LIN {X 0,Y 258.597,Z 623.646,A -85,B 0,C 180,E1 12291.002,E2 12291.002} C_VEL
LIN {X 0,Y 258.595,Z 623.557,A -85,B 0,C 180,E1 12285.987,E2 12285.987} C_VEL
LIN {X 0,Y 258.598,Z 623.543,A -85,B 0,C 180,E1 12281.064,E2 12281.064} C_VEL
LIN {X 0,Y 258.584,Z 623.565,A -85,B 0,C 180,E1 12276.085,E2 12276.085} C_VEL
LIN {X 0,Y 258.602,Z 623.568,A -85,B 0,C 180,E1 12271.205,E2 12271.205} C_VEL
LIN {X 0,Y 258.582,Z 623.556,A -85,B 0,C 180,E1 12268.101,E2 12268.101} C_VEL
LIN {X 0,Y 257.589,Z 623.666,A -85,B 0,C 180,E1 12266.394,E2 12266.394} C_VEL
LIN {X 0,Y 253.564,Z 624.201,A -85,B 0,C 180,E1 12263.518,E2 12263.518} C_VEL
LIN {X 0,Y 250.876,Z 624.542,A -85,B 0,C 180,E1 12261.032,E2 12261.032} C_VEL
LIN {X 0,Y 250.652,Z 624.55,A -85,B 0,C 180,E1 12260.264,E2 12260.264} C_VEL
LIN {X 0,Y 250.638,Z 624.544,A -85,B 0,C 180,E1 12255.113,E2 12255.113} C_VEL
LIN {X 0,Y 250.648,Z 624.524,A -85,B 0,C 180,E1 12250.342,E2 12250.342} C_VEL
LIN {X 0,Y 250.644,Z 624.566,A -85,B 0,C 180,E1 12245.494,E2 12245.494} C_VEL
LIN {X 0,Y 250.628,Z 624.52,A -85,B 0,C 180,E1 12240.458,E2 12240.458} C_VEL
LIN {X 0,Y 250.65,Z 624.566,A -85,B 0,C 180,E1 12235.654,E2 12235.654} C_VEL
LIN {X 0,Y 250.632,Z 624.544,A -85,B 0,C 180,E1 12230.818,E2 12230.818} C_VEL
LIN {X 0,Y 250.633,Z 624.535,A -85,B 0,C 180,E1 12225.68,E2 12225.68} C_VEL
LIN {X 0,Y 250.649,Z 624.552,A -85,B 0,C 180,E1 12220.907,E2 12220.907} C_VEL
LIN {X 0,Y 250.696,Z 624.842,A -85,B 0,C 180,E1 12216.993,E2 12216.993} C_VEL
LIN {X 0,Y 252.089,Z 628.267,A -85,B 0,C 180,E1 12215.389,E2 12215.389} C_VEL
LIN {X 0,Y 254.847,Z 634.454,A -85,B 0,C 180,E1 12212.676,E2 12212.676} C_VEL
LIN {X 0,Y 258.104,Z 641.784,A -85,B 0,C 180,E1 12209.755,E2 12209.755} C_VEL
LIN {X 0,Y 262.755,Z 653.333,A -85,B 0,C 180,E1 12205.724,E2 12205.724} C_VEL
LIN {X 0,Y 267.612,Z 666.638,A -85,B 0,C 180,E1 12201.686,E2 12201.686} C_VEL
LIN {X 0,Y 272.477,Z 681.722,A -85,B 0,C 180,E1 12197.674,E2 12197.674} C_VEL
LIN {X 0,Y 276.843,Z 696.584,A -85,B 0,C 180,E1 12194.192,E2 12194.192} C_VEL
LIN {X 0,Y 277.945,Z 699.592,A -85,B 0,C 180,E1 12193.916,E2 12193.916} C_VEL
LIN {X 0,Y 280.409,Z 735.71,A -85,B 0,C 180,E1 12192.492,E2 12192.492} C_VEL
LIN {X 0,Y 274.524,Z 880.829,A -85,B 0,C 180,E1 12188.924,E2 12188.924} C_VEL
LIN {X 0,Y 272.889,Z 899.096,A -85,B 0,C 180,E1 12188.126,E2 12188.126} C_VEL
LIN {X 0,Y 270.464,Z 916.83,A -85,B 0,C 180,E1 12186.989,E2 12186.989} C_VEL
LIN {X 0,Y 267.613,Z 933.578,A -85,B 0,C 180,E1 12185.52,E2 12185.52} C_VEL
LIN {X 0,Y 264.399,Z 949.953,A -85,B 0,C 180,E1 12183.643,E2 12183.643} C_VEL
LIN {X 0,Y 261.059,Z 965.272,A -85,B 0,C 180,E1 12181.392,E2 12181.392} C_VEL
LIN {X 0,Y 257.748,Z 979.594,A -85,B 0,C 180,E1 12178.753,E2 12178.753} C_VEL
LIN {X 0,Y 254.838,Z 992.418,A -85,B 0,C 180,E1 12175.818,E2 12175.818} C_VEL
LIN {X 0,Y 252.413,Z 1003.822,A -85,B 0,C 180,E1 12172.597,E2 12172.597} C_VEL
LIN {X 0,Y 250.561,Z 1014.181,A -85,B 0,C 180,E1 12168.961,E2 12168.961} C_VEL
LIN {X 0,Y 249.527,Z 1022.832,A -85,B 0,C 180,E1 12165.098,E2 12165.098} C_VEL
LIN {X 0,Y 249.297,Z 1029.658,A -85,B 0,C 180,E1 12161.1,E2 12161.1} C_VEL
LIN {X 0,Y 249.718,Z 1034.566,A -85,B 0,C 180,E1 12157.131,E2 12157.131} C_VEL
LIN {X 0,Y 250.306,Z 1037.499,A -85,B 0,C 180,E1 12153.436,E2 12153.436} C_VEL
LIN {X 0,Y 250.553,Z 1038.736,A -85,B 0,C 180,E1 12150.229,E2 12150.229} C_VEL
LIN {X 0,Y 250.237,Z 1038.662,A -85,B 0,C 180,E1 12147.023,E2 12147.023} C_VEL
LIN {X 0,Y 249.542,Z 1037.152,A -85,B 0,C 180,E1 12143.328,E2 12143.328} C_VEL
LIN {X 0,Y 249.014,Z 1033.682,A -85,B 0,C 180,E1 12139.122,E2 12139.122} C_VEL
LIN {X 0,Y 249.277,Z 1028.364,A -85,B 0,C 180,E1 12134.888,E2 12134.888} C_VEL
LIN {X 0,Y 250.59,Z 1021.098,A -85,B 0,C 180,E1 12130.66,E2 12130.66} C_VEL
LIN {X 0,Y 252.967,Z 1012.227,A -85,B 0,C 180,E1 12126.719,E2 12126.719} C_VEL
LIN {X 0,Y 256.245,Z 1001.804,A -85,B 0,C 180,E1 12123.088,E2 12123.088} C_VEL
LIN {X 0,Y 260.249,Z 989.873,A -85,B 0,C 180,E1 12119.782,E2 12119.782} C_VEL
LIN {X 0,Y 264.844,Z 976.404,A -85,B 0,C 180,E1 12116.81,E2 12116.81} C_VEL
LIN {X 0,Y 269.617,Z 961.83,A -85,B 0,C 180,E1 12114.262,E2 12114.262} C_VEL
LIN {X 0,Y 274.079,Z 946.842,A -85,B 0,C 180,E1 12112.203,E2 12112.203} C_VEL
LIN {X 0,Y 278.266,Z 930.98,A -85,B 0,C 180,E1 12110.507,E2 12110.507} C_VEL
LIN {X 0,Y 281.956,Z 914.615,A -85,B 0,C 180,E1 12109.177,E2 12109.177} C_VEL
LIN {X 0,Y 285.181,Z 896.361,A -85,B 0,C 180,E1 12108.103,E2 12108.103} C_VEL
LIN {X 0,Y 287.282,Z 878.288,A -85,B 0,C 180,E1 12107.378,E2 12107.378} C_VEL
LIN {X 0,Y 294.855,Z 735.141,A -85,B 0,C 180,E1 12103.879,E2 12103.879} C_VEL
LIN {X 0,Y 293.346,Z 713.913,A -85,B 0,C 180,E1 12102.776,E2 12102.776} C_VEL
LIN {X 0,Y 285.827,Z 700.894,A -85,B 0,C 180,E1 12100.524,E2 12100.524} C_VEL
LIN {X 0,Y 284.004,Z 697.557,A -85,B 0,C 180,E1 12099.847,E2 12099.847} C_VEL
LIN {X 0,Y 280.732,Z 687.562,A -85,B 0,C 180,E1 12096.244,E2 12096.244} C_VEL
LIN {X 0,Y 277.511,Z 678.838,A -85,B 0,C 180,E1 12092.468,E2 12092.468} C_VEL
LIN {X 0,Y 274.441,Z 671.373,A -85,B 0,C 180,E1 12088.507,E2 12088.507} C_VEL
LIN {X 0,Y 272.653,Z 667.299,A -85,B 0,C 180,E1 12085.873,E2 12085.873} C_VEL
LIN {X 0,Y 270.968,Z 663.499,A -85,B 0,C 180,E1 12083.025,E2 12083.025} C_VEL
LIN {X 0,Y 269.193,Z 659.526,A -85,B 0,C 180,E1 12079.303,E2 12079.303} C_VEL
LIN {X 0,Y 267.286,Z 655.366,A -85,B 0,C 180,E1 12073.19,E2 12073.19} C_VEL
LIN {X 0,Y 266.339,Z 654.288,A -85,B 0,C 180,E1 12067.984,E2 12067.984} C_VEL
LIN {X 0,Y 266.635,Z 654.723,A -85,B 0,C 180,E1 12062.579,E2 12062.579} C_VEL
LIN {X 0,Y 266.962,Z 655.866,A -85,B 0,C 180,E1 12059.962,E2 12059.962} C_VEL
LIN {X 0,Y 268.425,Z 659.327,A -85,B 0,C 180,E1 12054.656,E2 12054.656} C_VEL
LIN {X 0,Y 269.903,Z 663.428,A -85,B 0,C 180,E1 12050.619,E2 12050.619} C_VEL
LIN {X 0,Y 271.407,Z 667.48,A -85,B 0,C 180,E1 12047.446,E2 12047.446} C_VEL
LIN {X 0,Y 273.368,Z 672.921,A -85,B 0,C 180,E1 12043.86,E2 12043.86} C_VEL
LIN {X 0,Y 275.849,Z 680.778,A -85,B 0,C 180,E1 12039.636,E2 12039.636} C_VEL
LIN {X 0,Y 278.125,Z 689.309,A -85,B 0,C 180,E1 12035.805,E2 12035.805} C_VEL
LIN {X 0,Y 280.305,Z 698.744,A -85,B 0,C 180,E1 12032.141,E2 12032.141} C_VEL
LIN {X 0,Y 281.378,Z 704.237,A -85,B 0,C 180,E1 12030.283,E2 12030.283} C_VEL
LIN {X 0,Y 283.3,Z 708.755,A -85,B 0,C 180,E1 12029.527,E2 12029.527} C_VEL
LIN {X 0,Y 288.128,Z 736.946,A -85,B 0,C 180,E1 12027.253,E2 12027.253} C_VEL
LIN {X 0,Y 291.127,Z 758.877,A -85,B 0,C 180,E1 12025.756,E2 12025.756} C_VEL
LIN {X 0,Y 286.062,Z 844.009,A -85,B 0,C 180,E1 12023.499,E2 12023.499} C_VEL
LIN {X 0,Y 284.468,Z 860.29,A -85,B 0,C 180,E1 12022.719,E2 12022.719} C_VEL
LIN {X 0,Y 282.179,Z 875.724,A -85,B 0,C 180,E1 12021.636,E2 12021.636} C_VEL
LIN {X 0,Y 279.377,Z 889.681,A -85,B 0,C 180,E1 12020.305,E2 12020.305} C_VEL
LIN {X 0,Y 275.715,Z 904.283,A -85,B 0,C 180,E1 12018.476,E2 12018.476} C_VEL
LIN {X 0,Y 271.915,Z 916.881,A -85,B 0,C 180,E1 12016.418,E2 12016.418} C_VEL
LIN {X 0,Y 267.871,Z 928.54,A -85,B 0,C 180,E1 12013.969,E2 12013.969} C_VEL
LIN {X 0,Y 264.264,Z 937.852,A -85,B 0,C 180,E1 12011.462,E2 12011.462} C_VEL
LIN {X 0,Y 260.539,Z 946.484,A -85,B 0,C 180,E1 12008.44,E2 12008.44} C_VEL
LIN {X 0,Y 257.45,Z 953.125,A -85,B 0,C 180,E1 12005.355,E2 12005.355} C_VEL
LIN {X 0,Y 254.832,Z 958.272,A -85,B 0,C 180,E1 12001.984,E2 12001.984} C_VEL
LIN {X 0,Y 252.819,Z 961.87,A -85,B 0,C 180,E1 11998.332,E2 11998.332} C_VEL
LIN {X 0,Y 251.55,Z 963.593,A -85,B 0,C 180,E1 11994.667,E2 11994.667} C_VEL
LIN {X 0,Y 250.899,Z 963.561,A -85,B 0,C 180,E1 11990.773,E2 11990.773} C_VEL
LIN {X 0,Y 250.843,Z 961.794,A -85,B 0,C 180,E1 11987.155,E2 11987.155} C_VEL
LIN {X 0,Y 251.363,Z 958.066,A -85,B 0,C 180,E1 11983.339,E2 11983.339} C_VEL
LIN {X 0,Y 252.439,Z 952.682,A -85,B 0,C 180,E1 11979.806,E2 11979.806} C_VEL
LIN {X 0,Y 254.153,Z 945.316,A -85,B 0,C 180,E1 11976.324,E2 11976.324} C_VEL
LIN {X 0,Y 256.173,Z 936.954,A -85,B 0,C 180,E1 11973.356,E2 11973.356} C_VEL
LIN {X 0,Y 258.7,Z 926.457,A -85,B 0,C 180,E1 11970.442,E2 11970.442} C_VEL
LIN {X 0,Y 261.296,Z 914.754,A -85,B 0,C 180,E1 11967.916,E2 11967.916} C_VEL
LIN {X 0,Y 263.863,Z 902.135,A -85,B 0,C 180,E1 11965.762,E2 11965.762} C_VEL
LIN {X 0,Y 266.263,Z 888.571,A -85,B 0,C 180,E1 11963.964,E2 11963.964} C_VEL
LIN {X 0,Y 268.488,Z 873.21,A -85,B 0,C 180,E1 11962.403,E2 11962.403} C_VEL
LIN {X 0,Y 270.208,Z 856.922,A -85,B 0,C 180,E1 11961.22,E2 11961.22} C_VEL
LIN {X 0,Y 271.313,Z 840.68,A -85,B 0,C 180,E1 11960.434,E2 11960.434} C_VEL
LIN {X 0,Y 274.974,Z 752.221,A -85,B 0,C 180,E1 11958.038,E2 11958.038} C_VEL
LIN {X 0,Y 268.26,Z 704.82,A -85,B 0,C 180,E1 11955.593,E2 11955.593} C_VEL
LIN {X 0,Y 271.256,Z 690.293,A -85,B 0,C 180,E1 11952.628,E2 11952.628} C_VEL
LIN {X 0,Y 268.027,Z 675.976,A -85,B 0,C 180,E1 11948.556,E2 11948.556} C_VEL
LIN {X 0,Y 264.388,Z 662.466,A -85,B 0,C 180,E1 11944.328,E2 11944.328} C_VEL
LIN {X 0,Y 260.817,Z 651.102,A -85,B 0,C 180,E1 11940.361,E2 11940.361} C_VEL
LIN {X 0,Y 257.384,Z 641.549,A -85,B 0,C 180,E1 11936.639,E2 11936.639} C_VEL
LIN {X 0,Y 253.897,Z 632.375,A -85,B 0,C 180,E1 11932.665,E2 11932.665} C_VEL
LIN {X 0,Y 251.497,Z 627.253,A -85,B 0,C 180,E1 11930.113,E2 11930.113} C_VEL
LIN {X 0,Y 250.667,Z 624.683,A -85,B 0,C 180,E1 11928.733,E2 11928.733} C_VEL
LIN {X 0,Y 250.66,Z 624.573,A -85,B 0,C 180,E1 11923.78,E2 11923.78} C_VEL
LIN {X 0,Y 250.658,Z 624.548,A -85,B 0,C 180,E1 11918.935,E2 11918.935} C_VEL
LIN {X 0,Y 250.642,Z 624.527,A -85,B 0,C 180,E1 11913.925,E2 11913.925} C_VEL
LIN {X 0,Y 250.67,Z 624.564,A -85,B 0,C 180,E1 11909.12,E2 11909.12} C_VEL
LIN {X 0,Y 250.644,Z 624.533,A -85,B 0,C 180,E1 11904.261,E2 11904.261} C_VEL
LIN {X 0,Y 250.652,Z 624.55,A -85,B 0,C 180,E1 11900.264,E2 11900.264} C_VEL
LIN {X 0,Y 249.627,Z 624.66,A -85,B 0,C 180,E1 11898.503,E2 11898.503} C_VEL
LIN {X 0,Y 245.576,Z 625.199,A -85,B 0,C 180,E1 11895.536,E2 11895.536} C_VEL
LIN {X 0,Y 242.916,Z 625.539,A -85,B 0,C 180,E1 11892.968,E2 11892.968} C_VEL
LIN {X 0,Y 242.714,Z 625.55,A -85,B 0,C 180,E1 11892.174,E2 11892.174} C_VEL
LIN {X 0,Y 242.693,Z 625.518,A -85,B 0,C 180,E1 11887.1,E2 11887.1} C_VEL
LIN {X 0,Y 242.706,Z 625.517,A -85,B 0,C 180,E1 11882.125,E2 11882.125} C_VEL
LIN {X 0,Y 242.7,Z 625.559,A -85,B 0,C 180,E1 11877.167,E2 11877.167} C_VEL
LIN {X 0,Y 242.694,Z 625.517,A -85,B 0,C 180,E1 11871.948,E2 11871.948} C_VEL
LIN {X 0,Y 242.71,Z 625.533,A -85,B 0,C 180,E1 11867.147,E2 11867.147} C_VEL
LIN {X 0,Y 242.691,Z 625.567,A -85,B 0,C 180,E1 11862.121,E2 11862.121} C_VEL
LIN {X 0,Y 242.738,Z 625.842,A -85,B 0,C 180,E1 11859.569,E2 11859.569} C_VEL
LIN {X 0,Y 244.334,Z 629.512,A -85,B 0,C 180,E1 11857.631,E2 11857.631} C_VEL
LIN {X 0,Y 246.974,Z 635.346,A -85,B 0,C 180,E1 11854.844,E2 11854.844} C_VEL
LIN {X 0,Y 250.086,Z 642.133,A -85,B 0,C 180,E1 11851.851,E2 11851.851} C_VEL
LIN {X 0,Y 254.761,Z 653.796,A -85,B 0,C 180,E1 11847.474,E2 11847.474} C_VEL
LIN {X 0,Y 259.213,Z 665.715,A -85,B 0,C 180,E1 11843.557,E2 11843.557} C_VEL
LIN {X 0,Y 263.95,Z 679.981,A -85,B 0,C 180,E1 11839.485,E2 11839.485} C_VEL
LIN {X 0,Y 268.677,Z 695.94,A -85,B 0,C 180,E1 11835.454,E2 11835.454} C_VEL
LIN {X 0,Y 269.769,Z 698.685,A -85,B 0,C 180,E1 11835.085,E2 11835.085} C_VEL
LIN {X 0,Y 271.395,Z 702.547,A -85,B 0,C 180,E1 11834.732,E2 11834.732} C_VEL
LIN {X 0,Y 273.61,Z 736.548,A -85,B 0,C 180,E1 11833.358,E2 11833.358} C_VEL
LIN {X 0,Y 267.543,Z 880.121,A -85,B 0,C 180,E1 11829.757,E2 11829.757} C_VEL
LIN {X 0,Y 265.861,Z 898.397,A -85,B 0,C 180,E1 11828.943,E2 11828.943} C_VEL
LIN {X 0,Y 263.304,Z 916.451,A -85,B 0,C 180,E1 11827.759,E2 11827.759} C_VEL
LIN {X 0,Y 260.322,Z 933.306,A -85,B 0,C 180,E1 11826.238,E2 11826.238} C_VEL
LIN {X 0,Y 257.033,Z 949.39,A -85,B 0,C 180,E1 11824.337,E2 11824.337} C_VEL
LIN {X 0,Y 253.576,Z 964.616,A -85,B 0,C 180,E1 11822.033,E2 11822.033} C_VEL
LIN {X 0,Y 250.132,Z 978.897,A -85,B 0,C 180,E1 11819.32,E2 11819.32} C_VEL
LIN {X 0,Y 247.002,Z 992.117,A -85,B 0,C 180,E1 11816.183,E2 11816.183} C_VEL
LIN {X 0,Y 244.504,Z 1003.394,A -85,B 0,C 180,E1 11812.861,E2 11812.861} C_VEL
LIN {X 0,Y 242.657,Z 1013.28,A -85,B 0,C 180,E1 11809.247,E2 11809.247} C_VEL
LIN {X 0,Y 241.594,Z 1021.695,A -85,B 0,C 180,E1 11805.358,E2 11805.358} C_VEL
LIN {X 0,Y 241.341,Z 1028.525,A -85,B 0,C 180,E1 11801.229,E2 11801.229} C_VEL
LIN {X 0,Y 241.743,Z 1033.199,A -85,B 0,C 180,E1 11797.367,E2 11797.367} C_VEL
LIN {X 0,Y 242.371,Z 1036.215,A -85,B 0,C 180,E1 11793.548,E2 11793.548} C_VEL
LIN {X 0,Y 242.65,Z 1037.49,A -85,B 0,C 180,E1 11790.237,E2 11790.237} C_VEL
LIN {X 0,Y 242.298,Z 1037.466,A -85,B 0,C 180,E1 11786.925,E2 11786.925} C_VEL
LIN {X 0,Y 241.553,Z 1035.998,A -85,B 0,C 180,E1 11783.106,E2 11783.106} C_VEL
LIN {X 0,Y 241.028,Z 1032.576,A -85,B 0,C 180,E1 11778.757,E2 11778.757} C_VEL
LIN {X 0,Y 241.377,Z 1027.303,A -85,B 0,C 180,E1 11774.381,E2 11774.381} C_VEL
LIN {X 0,Y 242.847,Z 1020.08,A -85,B 0,C 180,E1 11770.018,E2 11770.018} C_VEL
LIN {X 0,Y 245.429,Z 1011.278,A -85,B 0,C 180,E1 11765.959,E2 11765.959} C_VEL
LIN {X 0,Y 248.944,Z 1000.915,A -85,B 0,C 180,E1 11762.232,E2 11762.232} C_VEL
LIN {X 0,Y 253.202,Z 989.077,A -85,B 0,C 180,E1 11758.849,E2 11758.849} C_VEL
LIN {X 0,Y 258.054,Z 975.679,A -85,B 0,C 180,E1 11755.819,E2 11755.819} C_VEL
LIN {X 0,Y 262.846,Z 961.787,A -85,B 0,C 180,E1 11753.329,E2 11753.329} C_VEL
LIN {X 0,Y 267.494,Z 947.056,A -85,B 0,C 180,E1 11751.238,E2 11751.238} C_VEL
LIN {X 0,Y 271.841,Z 931.515,A -85,B 0,C 180,E1 11749.52,E2 11749.52} C_VEL
LIN {X 0,Y 275.737,Z 915.143,A -85,B 0,C 180,E1 11748.148,E2 11748.148} C_VEL
LIN {X 0,Y 279.04,Z 897.565,A -85,B 0,C 180,E1 11747.076,E2 11747.076} C_VEL
LIN {X 0,Y 281.38,Z 879.001,A -85,B 0,C 180,E1 11746.298,E2 11746.298} C_VEL
LIN {X 0,Y 283.499,Z 842.829,A -85,B 0,C 180,E1 11745.373,E2 11745.373} C_VEL
LIN {X 0,Y 289.419,Z 736.279,A -85,B 0,C 180,E1 11742.745,E2 11742.745} C_VEL
LIN {X 0,Y 288.201,Z 717.926,A -85,B 0,C 180,E1 11741.767,E2 11741.767} C_VEL
LIN {X 0,Y 280.288,Z 704.05,A -85,B 0,C 180,E1 11739.252,E2 11739.252} C_VEL
LIN {X 0,Y 276.518,Z 697.804,A -85,B 0,C 180,E1 11737.831,E2 11737.831} C_VEL
LIN {X 0,Y 273.304,Z 688.322,A -85,B 0,C 180,E1 11734.037,E2 11734.037} C_VEL
LIN {X 0,Y 270.315,Z 680.495,A -85,B 0,C 180,E1 11730.201,E2 11730.201} C_VEL
LIN {X 0,Y 267.774,Z 674.014,A -85,B 0,C 180,E1 11726.343,E2 11726.343} C_VEL
LIN {X 0,Y 265.6,Z 669.326,A -85,B 0,C 180,E1 11722.734,E2 11722.734} C_VEL
LIN {X 0,Y 263.921,Z 665.479,A -85,B 0,C 180,E1 11719.014,E2 11719.014} C_VEL
LIN {X 0,Y 262.121,Z 661.451,A -85,B 0,C 180,E1 11713.006,E2 11713.006} C_VEL
LIN {X 0,Y 261.19,Z 660.419,A -85,B 0,C 180,E1 11707.699,E2 11707.699} C_VEL
LIN {X 0,Y 261.503,Z 660.871,A -85,B 0,C 180,E1 11702.41,E2 11702.41} C_VEL
LIN {X 0,Y 261.784,Z 662.197,A -85,B 0,C 180,E1 11699.562,E2 11699.562} C_VEL
LIN {X 0,Y 263.055,Z 665.27,A -85,B 0,C 180,E1 11694.766,E2 11694.766} C_VEL
LIN {X 0,Y 264.418,Z 669.141,A -85,B 0,C 180,E1 11690.861,E2 11690.861} C_VEL
LIN {X 0,Y 265.807,Z 673.148,A -85,B 0,C 180,E1 11687.619,E2 11687.619} C_VEL
LIN {X 0,Y 267.58,Z 678.248,A -85,B 0,C 180,E1 11684.17,E2 11684.17} C_VEL
LIN {X 0,Y 269.926,Z 686.085,A -85,B 0,C 180,E1 11679.849,E2 11679.849} C_VEL
LIN {X 0,Y 272.082,Z 694.639,A -85,B 0,C 180,E1 11675.926,E2 11675.926} C_VEL
LIN {X 0,Y 274.146,Z 703.986,A -85,B 0,C 180,E1 11672.288,E2 11672.288} C_VEL
LIN {X 0,Y 278.578,Z 712.773,A -85,B 0,C 180,E1 11670.576,E2 11670.576} C_VEL
LIN {X 0,Y 283.059,Z 740.327,A -85,B 0,C 180,E1 11668.302,E2 11668.302} C_VEL
LIN {X 0,Y 285.641,Z 760.611,A -85,B 0,C 180,E1 11666.891,E2 11666.891} C_VEL
LIN {X 0,Y 280.42,Z 844.7,A -85,B 0,C 180,E1 11664.638,E2 11664.638} C_VEL
LIN {X 0,Y 278.743,Z 861.013,A -85,B 0,C 180,E1 11663.847,E2 11663.847} C_VEL
LIN {X 0,Y 276.339,Z 876.45,A -85,B 0,C 180,E1 11662.751,E2 11662.751} C_VEL
LIN {X 0,Y 273.247,Z 891.044,A -85,B 0,C 180,E1 11661.333,E2 11661.333} C_VEL
LIN {X 0,Y 269.472,Z 905.321,A -85,B 0,C 180,E1 11659.508,E2 11659.508} C_VEL
LIN {X 0,Y 265.498,Z 917.826,A -85,B 0,C 180,E1 11657.43,E2 11657.43} C_VEL
LIN {X 0,Y 261.197,Z 929.61,A -85,B 0,C 180,E1 11654.912,E2 11654.912} C_VEL
LIN {X 0,Y 257.246,Z 939.243,A -85,B 0,C 180,E1 11652.253,E2 11652.253} C_VEL
LIN {X 0,Y 253.322,Z 947.821,A -85,B 0,C 180,E1 11649.162,E2 11649.162} C_VEL
LIN {X 0,Y 250.053,Z 954.415,A -85,B 0,C 180,E1 11646,E2 11646} C_VEL
LIN {X 0,Y 247.261,Z 959.53,A -85,B 0,C 180,E1 11642.535,E2 11642.535} C_VEL
LIN {X 0,Y 245.063,Z 963.168,A -85,B 0,C 180,E1 11638.692,E2 11638.692} C_VEL
LIN {X 0,Y 243.71,Z 964.821,A -85,B 0,C 180,E1 11634.947,E2 11634.947} C_VEL
LIN {X 0,Y 242.997,Z 964.762,A -85,B 0,C 180,E1 11630.925,E2 11630.925} C_VEL
LIN {X 0,Y 242.917,Z 963.009,A -85,B 0,C 180,E1 11627.238,E2 11627.238} C_VEL
LIN {X 0,Y 243.451,Z 959.239,A -85,B 0,C 180,E1 11623.251,E2 11623.251} C_VEL
LIN {X 0,Y 244.551,Z 953.938,A -85,B 0,C 180,E1 11619.65,E2 11619.65} C_VEL
LIN {X 0,Y 246.336,Z 946.564,A -85,B 0,C 180,E1 11616.04,E2 11616.04} C_VEL
LIN {X 0,Y 248.423,Z 938.304,A -85,B 0,C 180,E1 11612.999,E2 11612.999} C_VEL
LIN {X 0,Y 251.042,Z 927.866,A -85,B 0,C 180,E1 11610,E2 11610} C_VEL
LIN {X 0,Y 253.744,Z 916.28,A -85,B 0,C 180,E1 11607.402,E2 11607.402} C_VEL
LIN {X 0,Y 256.545,Z 903.091,A -85,B 0,C 180,E1 11605.081,E2 11605.081} C_VEL
LIN {X 0,Y 259.046,Z 889.548,A -85,B 0,C 180,E1 11603.239,E2 11603.239} C_VEL
LIN {X 0,Y 261.363,Z 874.224,A -85,B 0,C 180,E1 11601.641,E2 11601.641} C_VEL
LIN {X 0,Y 263.149,Z 858.159,A -85,B 0,C 180,E1 11600.438,E2 11600.438} C_VEL
LIN {X 0,Y 264.344,Z 841.574,A -85,B 0,C 180,E1 11599.606,E2 11599.606} C_VEL
LIN {X 0,Y 268.14,Z 753.168,A -85,B 0,C 180,E1 11597.16,E2 11597.16} C_VEL
LIN {X 0,Y 261.435,Z 704.987,A -85,B 0,C 180,E1 11594.599,E2 11594.599} C_VEL
LIN {X 0,Y 262.769,Z 698.408,A -85,B 0,C 180,E1 11593.304,E2 11593.304} C_VEL
LIN {X 0,Y 263.977,Z 692.922,A -85,B 0,C 180,E1 11592.133,E2 11592.133} C_VEL
LIN {X 0,Y 260.89,Z 678.952,A -85,B 0,C 180,E1 11588.044,E2 11588.044} C_VEL
LIN {X 0,Y 257.331,Z 665.522,A -85,B 0,C 180,E1 11583.707,E2 11583.707} C_VEL
LIN {X 0,Y 253.626,Z 653.753,A -85,B 0,C 180,E1 11579.432,E2 11579.432} C_VEL
LIN {X 0,Y 250.169,Z 643.88,A -85,B 0,C 180,E1 11575.42,E2 11575.42} C_VEL
LIN {X 0,Y 246.898,Z 635.905,A -85,B 0,C 180,E1 11571.712,E2 11571.712} C_VEL
LIN {X 0,Y 244.349,Z 629.521,A -85,B 0,C 180,E1 11568.478,E2 11568.478} C_VEL
LIN {X 0,Y 242.732,Z 625.669,A -85,B 0,C 180,E1 11566.209,E2 11566.209} C_VEL
LIN {X 0,Y 242.72,Z 625.52,A -85,B 0,C 180,E1 11561.074,E2 11561.074} C_VEL
LIN {X 0,Y 242.706,Z 625.539,A -85,B 0,C 180,E1 11556.094,E2 11556.094} C_VEL
LIN {X 0,Y 242.73,Z 625.546,A -85,B 0,C 180,E1 11550.992,E2 11550.992} C_VEL
LIN {X 0,Y 242.699,Z 625.508,A -85,B 0,C 180,E1 11545.894,E2 11545.894} C_VEL
LIN {X 0,Y 242.722,Z 625.548,A -85,B 0,C 180,E1 11540.749,E2 11540.749} C_VEL
LIN {X 0,Y 242.699,Z 625.518,A -85,B 0,C 180,E1 11535.778,E2 11535.778} C_VEL
LIN {X 0,Y 242.714,Z 625.55,A -85,B 0,C 180,E1 11532.174,E2 11532.174} C_VEL
LIN {X 0,Y 241.849,Z 625.639,A -85,B 0,C 180,E1 11530.484,E2 11530.484} C_VEL
LIN {X 0,Y 238.401,Z 626.094,A -85,B 0,C 180,E1 11527.806,E2 11527.806} C_VEL
LIN {X 0,Y 235.052,Z 626.521,A -85,B 0,C 180,E1 11524.771,E2 11524.771} C_VEL
LIN {X 0,Y 234.769,Z 626.539,A -85,B 0,C 180,E1 11523.813,E2 11523.813} C_VEL
LIN {X 0,Y 234.748,Z 626.514,A -85,B 0,C 180,E1 11518.536,E2 11518.536} C_VEL
LIN {X 0,Y 234.776,Z 626.502,A -85,B 0,C 180,E1 11513.398,E2 11513.398} C_VEL
LIN {X 0,Y 234.751,Z 626.542,A -85,B 0,C 180,E1 11508.204,E2 11508.204} C_VEL
LIN {X 0,Y 234.776,Z 626.571,A -85,B 0,C 180,E1 11503.167,E2 11503.167} C_VEL
LIN {X 0,Y 234.844,Z 627.105,A -85,B 0,C 180,E1 11502.405,E2 11502.405} C_VEL
LIN {X 0,Y 237.219,Z 632.279,A -85,B 0,C 180,E1 11499.346,E2 11499.346} C_VEL
LIN {X 0,Y 239.171,Z 636.504,A -85,B 0,C 180,E1 11497.121,E2 11497.121} C_VEL
LIN {X 0,Y 241.374,Z 641.447,A -85,B 0,C 180,E1 11494.744,E2 11494.744} C_VEL
LIN {X 0,Y 244.203,Z 647.836,A -85,B 0,C 180,E1 11491.911,E2 11491.911} C_VEL
LIN {X 0,Y 248.35,Z 658.225,A -85,B 0,C 180,E1 11487.898,E2 11487.898} C_VEL
LIN {X 0,Y 252.84,Z 670.501,A -85,B 0,C 180,E1 11483.778,E2 11483.778} C_VEL
LIN {X 0,Y 257.354,Z 684.492,A -85,B 0,C 180,E1 11479.694,E2 11479.694} C_VEL
LIN {X 0,Y 261.13,Z 697.26,A -85,B 0,C 180,E1 11476.432,E2 11476.432} C_VEL
LIN {X 0,Y 264.867,Z 705.427,A -85,B 0,C 180,E1 11475.581,E2 11475.581} C_VEL
LIN {X 0,Y 266.844,Z 737.351,A -85,B 0,C 180,E1 11474.256,E2 11474.256} C_VEL
LIN {X 0,Y 260.576,Z 879.607,A -85,B 0,C 180,E1 11470.617,E2 11470.617} C_VEL
LIN {X 0,Y 258.847,Z 897.838,A -85,B 0,C 180,E1 11469.786,E2 11469.786} C_VEL
LIN {X 0,Y 256.191,Z 915.969,A -85,B 0,C 180,E1 11468.571,E2 11468.571} C_VEL
LIN {X 0,Y 253.172,Z 932.478,A -85,B 0,C 180,E1 11467.048,E2 11467.048} C_VEL
LIN {X 0,Y 249.705,Z 948.809,A -85,B 0,C 180,E1 11465.072,E2 11465.072} C_VEL
LIN {X 0,Y 246.117,Z 963.992,A -85,B 0,C 180,E1 11462.706,E2 11462.706} C_VEL
LIN {X 0,Y 242.542,Z 978.199,A -85,B 0,C 180,E1 11459.922,E2 11459.922} C_VEL
LIN {X 0,Y 239.39,Z 990.916,A -85,B 0,C 180,E1 11456.814,E2 11456.814} C_VEL
LIN {X 0,Y 236.758,Z 1002.217,A -85,B 0,C 180,E1 11453.39,E2 11453.39} C_VEL
LIN {X 0,Y 234.802,Z 1012.118,A -85,B 0,C 180,E1 11449.659,E2 11449.659} C_VEL
LIN {X 0,Y 233.663,Z 1020.54,A -85,B 0,C 180,E1 11445.64,E2 11445.64} C_VEL
LIN {X 0,Y 233.386,Z 1027.373,A -85,B 0,C 180,E1 11441.366,E2 11441.366} C_VEL
LIN {X 0,Y 233.846,Z 1032.268,A -85,B 0,C 180,E1 11437.123,E2 11437.123} C_VEL
LIN {X 0,Y 234.513,Z 1035.165,A -85,B 0,C 180,E1 11433.178,E2 11433.178} C_VEL
LIN {X 0,Y 234.729,Z 1036.351,A -85,B 0,C 180,E1 11429.756,E2 11429.756} C_VEL
LIN {X 0,Y 234.261,Z 1036.177,A -85,B 0,C 180,E1 11426.33,E2 11426.33} C_VEL
LIN {X 0,Y 233.431,Z 1034.406,A -85,B 0,C 180,E1 11422.122,E2 11422.122} C_VEL
LIN {X 0,Y 233.047,Z 1030.736,A -85,B 0,C 180,E1 11417.613,E2 11417.613} C_VEL
LIN {X 0,Y 233.67,Z 1025.211,A -85,B 0,C 180,E1 11413.084,E2 11413.084} C_VEL
LIN {X 0,Y 235.399,Z 1018.167,A -85,B 0,C 180,E1 11408.836,E2 11408.836} C_VEL
LIN {X 0,Y 238.347,Z 1009.151,A -85,B 0,C 180,E1 11404.667,E2 11404.667} C_VEL
LIN {X 0,Y 242.251,Z 998.612,A -85,B 0,C 180,E1 11400.855,E2 11400.855} C_VEL
LIN {X 0,Y 246.904,Z 986.545,A -85,B 0,C 180,E1 11397.412,E2 11397.412} C_VEL
LIN {X 0,Y 251.992,Z 973.282,A -85,B 0,C 180,E1 11394.429,E2 11394.429} C_VEL
LIN {X 0,Y 257.037,Z 959.234,A -85,B 0,C 180,E1 11391.935,E2 11391.935} C_VEL
LIN {X 0,Y 261.956,Z 944.077,A -85,B 0,C 180,E1 11389.83,E2 11389.83} C_VEL
LIN {X 0,Y 266.55,Z 928.045,A -85,B 0,C 180,E1 11388.111,E2 11388.111} C_VEL
LIN {X 0,Y 270.646,Z 911.008,A -85,B 0,C 180,E1 11386.741,E2 11386.741} C_VEL
LIN {X 0,Y 273.902,Z 893.411,A -85,B 0,C 180,E1 11385.722,E2 11385.722} C_VEL
LIN {X 0,Y 276.085,Z 875.179,A -85,B 0,C 180,E1 11385.005,E2 11385.005} C_VEL
LIN {X 0,Y 284.098,Z 737.345,A -85,B 0,C 180,E1 11381.564,E2 11381.564} C_VEL
LIN {X 0,Y 283.153,Z 721.957,A -85,B 0,C 180,E1 11380.721,E2 11380.721} C_VEL
LIN {X 0,Y 276.319,Z 709.752,A -85,B 0,C 180,E1 11378.424,E2 11378.424} C_VEL
LIN {X 0,Y 269.165,Z 698.327,A -85,B 0,C 180,E1 11375.676,E2 11375.676} C_VEL
LIN {X 0,Y 266.21,Z 689.866,A -85,B 0,C 180,E1 11371.915,E2 11371.915} C_VEL
LIN {X 0,Y 263.35,Z 682.543,A -85,B 0,C 180,E1 11367.839,E2 11367.839} C_VEL
LIN {X 0,Y 261.62,Z 678.487,A -85,B 0,C 180,E1 11365.074,E2 11365.074} C_VEL
LIN {X 0,Y 260.333,Z 675.308,A -85,B 0,C 180,E1 11362.586,E2 11362.586} C_VEL
LIN {X 0,Y 258.749,Z 671.574,A -85,B 0,C 180,E1 11358.94,E2 11358.94} C_VEL
LIN {X 0,Y 256.984,Z 667.562,A -85,B 0,C 180,E1 11352.813,E2 11352.813} C_VEL
LIN {X 0,Y 256.072,Z 666.567,A -85,B 0,C 180,E1 11347.357,E2 11347.357} C_VEL
LIN {X 0,Y 256.422,Z 667.088,A -85,B 0,C 180,E1 11342.011,E2 11342.011} C_VEL
LIN {X 0,Y 257.691,Z 671.016,A -85,B 0,C 180,E1 11335.103,E2 11335.103} C_VEL
LIN {X 0,Y 258.972,Z 675.105,A -85,B 0,C 180,E1 11330.892,E2 11330.892} C_VEL
LIN {X 0,Y 260.222,Z 678.826,A -85,B 0,C 180,E1 11327.799,E2 11327.799} C_VEL
LIN {X 0,Y 261.927,Z 684.175,A -85,B 0,C 180,E1 11324.146,E2 11324.146} C_VEL
LIN {X 0,Y 264.009,Z 691.401,A -85,B 0,C 180,E1 11320.071,E2 11320.071} C_VEL
LIN {X 0,Y 266.146,Z 700.299,A -85,B 0,C 180,E1 11315.909,E2 11315.909} C_VEL
LIN {X 0,Y 267.11,Z 704.257,A -85,B 0,C 180,E1 11314.383,E2 11314.383} C_VEL
LIN {X 0,Y 273.705,Z 716.398,A -85,B 0,C 180,E1 11311.766,E2 11311.766} C_VEL
LIN {X 0,Y 274.402,Z 719.247,A -85,B 0,C 180,E1 11311.44,E2 11311.44} C_VEL
LIN {X 0,Y 278.53,Z 746.876,A -85,B 0,C 180,E1 11309.143,E2 11309.143} C_VEL
LIN {X 0,Y 280.276,Z 762.256,A -85,B 0,C 180,E1 11308.073,E2 11308.073} C_VEL
LIN {X 0,Y 274.892,Z 845.39,A -85,B 0,C 180,E1 11305.823,E2 11305.823} C_VEL
LIN {X 0,Y 273.132,Z 861.754,A -85,B 0,C 180,E1 11305.022,E2 11305.022} C_VEL
LIN {X 0,Y 270.508,Z 877.805,A -85,B 0,C 180,E1 11303.864,E2 11303.864} C_VEL
LIN {X 0,Y 267.252,Z 892.337,A -85,B 0,C 180,E1 11302.422,E2 11302.422} C_VEL
LIN {X 0,Y 263.364,Z 906.337,A -85,B 0,C 180,E1 11300.604,E2 11300.604} C_VEL
LIN {X 0,Y 259.135,Z 918.995,A -85,B 0,C 180,E1 11298.464,E2 11298.464} C_VEL
LIN {X 0,Y 254.653,Z 930.613,A -85,B 0,C 180,E1 11295.932,E2 11295.932} C_VEL
LIN {X 0,Y 250.632,Z 939.926,A -85,B 0,C 180,E1 11293.327,E2 11293.327} C_VEL
LIN {X 0,Y 246.442,Z 948.57,A -85,B 0,C 180,E1 11290.172,E2 11290.172} C_VEL
LIN {X 0,Y 242.687,Z 955.705,A -85,B 0,C 180,E1 11286.683,E2 11286.683} C_VEL
LIN {X 0,Y 239.533,Z 961.081,A -85,B 0,C 180,E1 11282.864,E2 11282.864} C_VEL
LIN {X 0,Y 237.274,Z 964.518,A -85,B 0,C 180,E1 11278.986,E2 11278.986} C_VEL
LIN {X 0,Y 235.761,Z 966.125,A -85,B 0,C 180,E1 11274.825,E2 11274.825} C_VEL
LIN {X 0,Y 235.082,Z 965.929,A -85,B 0,C 180,E1 11270.932,E2 11270.932} C_VEL
LIN {X 0,Y 235.018,Z 963.851,A -85,B 0,C 180,E1 11266.814,E2 11266.814} C_VEL
LIN {X 0,Y 235.575,Z 960.224,A -85,B 0,C 180,E1 11263,E2 11263} C_VEL
LIN {X 0,Y 236.761,Z 954.743,A -85,B 0,C 180,E1 11259.234,E2 11259.234} C_VEL
LIN {X 0,Y 238.499,Z 947.861,A -85,B 0,C 180,E1 11255.774,E2 11255.774} C_VEL
LIN {X 0,Y 240.677,Z 939.614,A -85,B 0,C 180,E1 11252.619,E2 11252.619} C_VEL
LIN {X 0,Y 243.394,Z 929.224,A -85,B 0,C 180,E1 11249.529,E2 11249.529} C_VEL
LIN {X 0,Y 246.207,Z 917.743,A -85,B 0,C 180,E1 11246.857,E2 11246.857} C_VEL
LIN {X 0,Y 249.135,Z 904.538,A -85,B 0,C 180,E1 11244.452,E2 11244.452} C_VEL
LIN {X 0,Y 251.709,Z 891.341,A -85,B 0,C 180,E1 11242.582,E2 11242.582} C_VEL
LIN {X 0,Y 254.156,Z 875.945,A -85,B 0,C 180,E1 11240.914,E2 11240.914} C_VEL
LIN {X 0,Y 256.032,Z 860.295,A -85,B 0,C 180,E1 11239.679,E2 11239.679} C_VEL
LIN {X 0,Y 257.371,Z 843.117,A -85,B 0,C 180,E1 11238.771,E2 11238.771} C_VEL
LIN {X 0,Y 261.466,Z 756.463,A -85,B 0,C 180,E1 11236.337,E2 11236.337} C_VEL
LIN {X 0,Y 255.462,Z 710.739,A -85,B 0,C 180,E1 11233.88,E2 11233.88} C_VEL
LIN {X 0,Y 254.685,Z 704.29,A -85,B 0,C 180,E1 11233.463,E2 11233.463} C_VEL
LIN {X 0,Y 256.716,Z 695.552,A -85,B 0,C 180,E1 11231.61,E2 11231.61} C_VEL
LIN {X 0,Y 253.776,Z 682.019,A -85,B 0,C 180,E1 11227.531,E2 11227.531} C_VEL
LIN {X 0,Y 250.551,Z 669.499,A -85,B 0,C 180,E1 11223.369,E2 11223.369} C_VEL
LIN {X 0,Y 246.77,Z 657.142,A -85,B 0,C 180,E1 11218.753,E2 11218.753} C_VEL
LIN {X 0,Y 243.458,Z 647.865,A -85,B 0,C 180,E1 11214.814,E2 11214.814} C_VEL
LIN {X 0,Y 239.947,Z 638.608,A -85,B 0,C 180,E1 11210.39,E2 11210.39} C_VEL
LIN {X 0,Y 236.538,Z 630.666,A -85,B 0,C 180,E1 11205.94,E2 11205.94} C_VEL
LIN {X 0,Y 234.794,Z 626.655,A -85,B 0,C 180,E1 11203.264,E2 11203.264} C_VEL
LIN {X 0,Y 234.769,Z 626.541,A -85,B 0,C 180,E1 11198.138,E2 11198.138} C_VEL
LIN {X 0,Y 234.778,Z 626.503,A -85,B 0,C 180,E1 11192.967,E2 11192.967} C_VEL
LIN {X 0,Y 234.764,Z 626.514,A -85,B 0,C 180,E1 11187.937,E2 11187.937} C_VEL
LIN {X 0,Y 234.788,Z 626.535,A -85,B 0,C 180,E1 11182.801,E2 11182.801} C_VEL
LIN {X 0,Y 234.755,Z 626.492,A -85,B 0,C 180,E1 11177.602,E2 11177.602} C_VEL
LIN {X 0,Y 234.775,Z 626.546,A -85,B 0,C 180,E1 11172.545,E2 11172.545} C_VEL
LIN {X 0,Y 234.756,Z 626.502,A -85,B 0,C 180,E1 11167.342,E2 11167.342} C_VEL
LIN {X 0,Y 234.769,Z 626.539,A -85,B 0,C 180,E1 11163.813,E2 11163.813} C_VEL
LIN {X 0,Y 233.897,Z 626.626,A -85,B 0,C 180,E1 11162.066,E2 11162.066} C_VEL
LIN {X 0,Y 230.463,Z 627.071,A -85,B 0,C 180,E1 11159.295,E2 11159.295} C_VEL
LIN {X 0,Y 227.116,Z 627.505,A -85,B 0,C 180,E1 11156.154,E2 11156.154} C_VEL
LIN {X 0,Y 226.82,Z 627.517,A -85,B 0,C 180,E1 11155.162,E2 11155.162} C_VEL
LIN {X 0,Y 226.821,Z 627.525,A -85,B 0,C 180,E1 11149.845,E2 11149.845} C_VEL
LIN {X 0,Y 226.852,Z 627.813,A -85,B 0,C 180,E1 11146.004,E2 11146.004} C_VEL
LIN {X 0,Y 228.721,Z 631.795,A -85,B 0,C 180,E1 11143.212,E2 11143.212} C_VEL
LIN {X 0,Y 231.382,Z 637.458,A -85,B 0,C 180,E1 11139.776,E2 11139.776} C_VEL
LIN {X 0,Y 233.571,Z 642.529,A -85,B 0,C 180,E1 11137.074,E2 11137.074} C_VEL
LIN {X 0,Y 236.529,Z 649.009,A -85,B 0,C 180,E1 11133.92,E2 11133.92} C_VEL
LIN {X 0,Y 240.51,Z 658.784,A -85,B 0,C 180,E1 11129.8,E2 11129.8} C_VEL
LIN {X 0,Y 244.964,Z 670.919,A -85,B 0,C 180,E1 11125.435,E2 11125.435} C_VEL
LIN {X 0,Y 249.314,Z 684.221,A -85,B 0,C 180,E1 11121.272,E2 11121.272} C_VEL
LIN {X 0,Y 253.275,Z 697.424,A -85,B 0,C 180,E1 11117.695,E2 11117.695} C_VEL
LIN {X 0,Y 258.394,Z 708.243,A -85,B 0,C 180,E1 11116.477,E2 11116.477} C_VEL
LIN {X 0,Y 260.144,Z 738.2,A -85,B 0,C 180,E1 11115.2,E2 11115.2} C_VEL
LIN {X 0,Y 253.674,Z 878.901,A -85,B 0,C 180,E1 11111.525,E2 11111.525} C_VEL
LIN {X 0,Y 251.89,Z 897.143,A -85,B 0,C 180,E1 11110.677,E2 11110.677} C_VEL
LIN {X 0,Y 249.244,Z 914.685,A -85,B 0,C 180,E1 11109.483,E2 11109.483} C_VEL
LIN {X 0,Y 245.992,Z 931.928,A -85,B 0,C 180,E1 11107.862,E2 11107.862} C_VEL
LIN {X 0,Y 242.42,Z 948.096,A -85,B 0,C 180,E1 11105.852,E2 11105.852} C_VEL
LIN {X 0,Y 238.69,Z 963.3,A -85,B 0,C 180,E1 11103.418,E2 11103.418} C_VEL
LIN {X 0,Y 234.981,Z 977.456,A -85,B 0,C 180,E1 11100.563,E2 11100.563} C_VEL
LIN {X 0,Y 231.584,Z 990.602,A -85,B 0,C 180,E1 11097.236,E2 11097.236} C_VEL
LIN {X 0,Y 228.865,Z 1001.788,A -85,B 0,C 180,E1 11093.699,E2 11093.699} C_VEL
LIN {X 0,Y 226.853,Z 1011.553,A -85,B 0,C 180,E1 11089.84,E2 11089.84} C_VEL
LIN {X 0,Y 225.695,Z 1019.829,A -85,B 0,C 180,E1 11085.679,E2 11085.679} C_VEL
LIN {X 0,Y 225.44,Z 1026.554,A -85,B 0,C 180,E1 11081.254,E2 11081.254} C_VEL
LIN {X 0,Y 225.955,Z 1031.337,A -85,B 0,C 180,E1 11076.862,E2 11076.862} C_VEL
LIN {X 0,Y 226.618,Z 1033.992,A -85,B 0,C 180,E1 11073.035,E2 11073.035} C_VEL
LIN {X 0,Y 226.826,Z 1035.1,A -85,B 0,C 180,E1 11069.748,E2 11069.748} C_VEL
LIN {X 0,Y 226.31,Z 1034.979,A -85,B 0,C 180,E1 11066.201,E2 11066.201} C_VEL
LIN {X 0,Y 225.43,Z 1033.251,A -85,B 0,C 180,E1 11061.841,E2 11061.841} C_VEL
LIN {X 0,Y 225.088,Z 1029.626,A -85,B 0,C 180,E1 11057.168,E2 11057.168} C_VEL
LIN {X 0,Y 225.829,Z 1024.158,A -85,B 0,C 180,E1 11052.478,E2 11052.478} C_VEL
LIN {X 0,Y 227.902,Z 1016.725,A -85,B 0,C 180,E1 11047.834,E2 11047.834} C_VEL
LIN {X 0,Y 231.163,Z 1007.648,A -85,B 0,C 180,E1 11043.544,E2 11043.544} C_VEL
LIN {X 0,Y 235.412,Z 997.038,A -85,B 0,C 180,E1 11039.641,E2 11039.641} C_VEL
LIN {X 0,Y 240.413,Z 984.886,A -85,B 0,C 180,E1 11036.131,E2 11036.131} C_VEL
LIN {X 0,Y 245.787,Z 971.635,A -85,B 0,C 180,E1 11033.128,E2 11033.128} C_VEL
LIN {X 0,Y 251.309,Z 956.899,A -85,B 0,C 180,E1 11030.52,E2 11030.52} C_VEL
LIN {X 0,Y 256.349,Z 942.01,A -85,B 0,C 180,E1 11028.466,E2 11028.466} C_VEL
LIN {X 0,Y 261.168,Z 925.715,A -85,B 0,C 180,E1 11026.742,E2 11026.742} C_VEL
LIN {X 0,Y 265.213,Z 909.272,A -85,B 0,C 180,E1 11025.441,E2 11025.441} C_VEL
LIN {X 0,Y 268.572,Z 891.452,A -85,B 0,C 180,E1 11024.426,E2 11024.426} C_VEL
LIN {X 0,Y 270.713,Z 873.229,A -85,B 0,C 180,E1 11023.732,E2 11023.732} C_VEL
LIN {X 0,Y 278.9,Z 738.276,A -85,B 0,C 180,E1 11020.331,E2 11020.331} C_VEL
LIN {X 0,Y 278.212,Z 725.906,A -85,B 0,C 180,E1 11019.636,E2 11019.636} C_VEL
LIN {X 0,Y 271.604,Z 714.193,A -85,B 0,C 180,E1 11017.27,E2 11017.27} C_VEL
LIN {X 0,Y 264.718,Z 703.383,A -85,B 0,C 180,E1 11014.57,E2 11014.57} C_VEL
LIN {X 0,Y 261.59,Z 698.338,A -85,B 0,C 180,E1 11013.067,E2 11013.067} C_VEL
LIN {X 0,Y 258.664,Z 690.431,A -85,B 0,C 180,E1 11008.893,E2 11008.893} C_VEL
LIN {X 0,Y 256.436,Z 684.705,A -85,B 0,C 180,E1 11005.15,E2 11005.15} C_VEL
LIN {X 0,Y 254.953,Z 681.101,A -85,B 0,C 180,E1 11002.252,E2 11002.252} C_VEL
LIN {X 0,Y 253.458,Z 677.5,A -85,B 0,C 180,E1 10998.634,E2 10998.634} C_VEL
LIN {X 0,Y 251.878,Z 673.728,A -85,B 0,C 180,E1 10992.844,E2 10992.844} C_VEL
LIN {X 0,Y 250.949,Z 672.711,A -85,B 0,C 180,E1 10987.325,E2 10987.325} C_VEL
LIN {X 0,Y 251.243,Z 673.183,A -85,B 0,C 180,E1 10982.052,E2 10982.052} C_VEL
LIN {X 0,Y 252.351,Z 676.98,A -85,B 0,C 180,E1 10975.227,E2 10975.227} C_VEL
LIN {X 0,Y 253.484,Z 680.809,A -85,B 0,C 180,E1 10971.15,E2 10971.15} C_VEL
LIN {X 0,Y 254.655,Z 684.52,A -85,B 0,C 180,E1 10967.989,E2 10967.989} C_VEL
LIN {X 0,Y 256.201,Z 689.684,A -85,B 0,C 180,E1 10964.378,E2 10964.378} C_VEL
LIN {X 0,Y 258.122,Z 696.803,A -85,B 0,C 180,E1 10960.268,E2 10960.268} C_VEL
LIN {X 0,Y 259.677,Z 703.406,A -85,B 0,C 180,E1 10957.114,E2 10957.114} C_VEL
LIN {X 0,Y 264.755,Z 712.597,A -85,B 0,C 180,E1 10954.708,E2 10954.708} C_VEL
LIN {X 0,Y 269.676,Z 721.74,A -85,B 0,C 180,E1 10952.703,E2 10952.703} C_VEL
LIN {X 0,Y 273.552,Z 749.322,A -85,B 0,C 180,E1 10950.342,E2 10950.342} C_VEL
LIN {X 0,Y 275.056,Z 763.735,A -85,B 0,C 180,E1 10949.306,E2 10949.306} C_VEL
LIN {X 0,Y 269.488,Z 846.081,A -85,B 0,C 180,E1 10947.056,E2 10947.056} C_VEL
LIN {X 0,Y 267.64,Z 862.497,A -85,B 0,C 180,E1 10946.245,E2 10946.245} C_VEL
LIN {X 0,Y 264.909,Z 878.493,A -85,B 0,C 180,E1 10945.082,E2 10945.082} C_VEL
LIN {X 0,Y 261.464,Z 893.232,A -85,B 0,C 180,E1 10943.607,E2 10943.607} C_VEL
LIN {X 0,Y 257.293,Z 907.563,A -85,B 0,C 180,E1 10941.719,E2 10941.719} C_VEL
LIN {X 0,Y 252.932,Z 919.981,A -85,B 0,C 180,E1 10939.585,E2 10939.585} C_VEL
LIN {X 0,Y 248.175,Z 931.701,A -85,B 0,C 180,E1 10936.99,E2 10936.99} C_VEL
LIN {X 0,Y 243.749,Z 941.377,A -85,B 0,C 180,E1 10934.214,E2 10934.214} C_VEL
LIN {X 0,Y 239.13,Z 950.35,A -85,B 0,C 180,E1 10930.816,E2 10930.816} C_VEL
LIN {X 0,Y 235.351,Z 957.03,A -85,B 0,C 180,E1 10927.396,E2 10927.396} C_VEL
LIN {X 0,Y 232.002,Z 962.342,A -85,B 0,C 180,E1 10923.479,E2 10923.479} C_VEL
LIN {X 0,Y 229.578,Z 965.749,A -85,B 0,C 180,E1 10919.481,E2 10919.481} C_VEL
LIN {X 0,Y 227.938,Z 967.342,A -85,B 0,C 180,E1 10915.182,E2 10915.182} C_VEL
LIN {X 0,Y 227.18,Z 967.12,A -85,B 0,C 180,E1 10911.083,E2 10911.083} C_VEL
LIN {X 0,Y 227.091,Z 965.06,A -85,B 0,C 180,E1 10906.893,E2 10906.893} C_VEL
LIN {X 0,Y 227.674,Z 961.334,A -85,B 0,C 180,E1 10902.85,E2 10902.85} C_VEL
LIN {X 0,Y 228.877,Z 955.979,A -85,B 0,C 180,E1 10899.048,E2 10899.048} C_VEL
LIN {X 0,Y 230.835,Z 948.571,A -85,B 0,C 180,E1 10895.218,E2 10895.218} C_VEL
LIN {X 0,Y 233.34,Z 939.464,A -85,B 0,C 180,E1 10891.718,E2 10891.718} C_VEL
LIN {X 0,Y 236.024,Z 929.65,A -85,B 0,C 180,E1 10888.771,E2 10888.771} C_VEL
LIN {X 0,Y 238.96,Z 918.07,A -85,B 0,C 180,E1 10886.041,E2 10886.041} C_VEL
LIN {X 0,Y 242.012,Z 904.855,A -85,B 0,C 180,E1 10883.595,E2 10883.595} C_VEL
LIN {X 0,Y 244.73,Z 891.317,A -85,B 0,C 180,E1 10881.66,E2 10881.66} C_VEL
LIN {X 0,Y 247.244,Z 876.023,A -85,B 0,C 180,E1 10879.985,E2 10879.985} C_VEL
LIN {X 0,Y 249.199,Z 860.027,A -85,B 0,C 180,E1 10878.721,E2 10878.721} C_VEL
LIN {X 0,Y 250.547,Z 843.121,A -85,B 0,C 180,E1 10877.825,E2 10877.825} C_VEL
LIN {X 0,Y 254.678,Z 755.368,A -85,B 0,C 180,E1 10875.295,E2 10875.295} C_VEL
LIN {X 0,Y 247.987,Z 704.116,A -85,B 0,C 180,E1 10872.337,E2 10872.337} C_VEL
LIN {X 0,Y 249.379,Z 697.734,A -85,B 0,C 180,E1 10870.927,E2 10870.927} C_VEL
LIN {X 0,Y 246.366,Z 683.659,A -85,B 0,C 180,E1 10866.523,E2 10866.523} C_VEL
LIN {X 0,Y 243.116,Z 671.131,A -85,B 0,C 180,E1 10862.158,E2 10862.158} C_VEL
LIN {X 0,Y 239.491,Z 659.272,A -85,B 0,C 180,E1 10857.495,E2 10857.495} C_VEL
LIN {X 0,Y 236.058,Z 649.733,A -85,B 0,C 180,E1 10853.183,E2 10853.183} C_VEL
LIN {X 0,Y 233.032,Z 642.198,A -85,B 0,C 180,E1 10849.293,E2 10849.293} C_VEL
LIN {X 0,Y 230.552,Z 635.908,A -85,B 0,C 180,E1 10845.691,E2 10845.691} C_VEL
LIN {X 0,Y 228.213,Z 631.107,A -85,B 0,C 180,E1 10842.433,E2 10842.433} C_VEL
LIN {X 0,Y 226.858,Z 627.615,A -85,B 0,C 180,E1 10839.724,E2 10839.724} C_VEL
LIN {X 0,Y 226.826,Z 627.492,A -85,B 0,C 180,E1 10834.481,E2 10834.481} C_VEL
LIN {X 0,Y 226.847,Z 627.527,A -85,B 0,C 180,E1 10829.223,E2 10829.223} C_VEL
LIN {X 0,Y 226.821,Z 627.5,A -85,B 0,C 180,E1 10823.926,E2 10823.926} C_VEL
LIN {X 0,Y 226.83,Z 627.485,A -85,B 0,C 180,E1 10818.771,E2 10818.771} C_VEL
LIN {X 0,Y 226.823,Z 627.543,A -85,B 0,C 180,E1 10813.511,E2 10813.511} C_VEL
LIN {X 0,Y 226.839,Z 627.478,A -85,B 0,C 180,E1 10808.109,E2 10808.109} C_VEL
LIN {X 0,Y 226.814,Z 627.504,A -85,B 0,C 180,E1 10802.78,E2 10802.78} C_VEL
LIN {X 0,Y 226.83,Z 627.516,A -85,B 0,C 180,E1 10797.727,E2 10797.727} C_VEL
LIN {X 0,Y 226.82,Z 627.517,A -85,B 0,C 180,E1 10795.162,E2 10795.162} C_VEL
LIN {X 0,Y 225.739,Z 627.631,A -85,B 0,C 180,E1 10793.853,E2 10793.853} C_VEL
LIN {X 0,Y 219.85,Z 628.683,A -85,B 0,C 180,E1 10790.651,E2 10790.651} C_VEL
LIN {X 0,Y 219.151,Z 629.692,A -85,B 0,C 180,E1 10789.53,E2 10789.53} C_VEL
LIN {X 0,Y 219.196,Z 629.928,A -85,B 0,C 180,E1 10789.346,E2 10789.346} C_VEL
LIN {X 0,Y 221.411,Z 634.05,A -85,B 0,C 180,E1 10785.886,E2 10785.886} C_VEL
LIN {X 0,Y 223.519,Z 638.442,A -85,B 0,C 180,E1 10782.829,E2 10782.829} C_VEL
LIN {X 0,Y 225.724,Z 643.236,A -85,B 0,C 180,E1 10779.898,E2 10779.898} C_VEL
LIN {X 0,Y 228.929,Z 650.377,A -85,B 0,C 180,E1 10776.035,E2 10776.035} C_VEL
LIN {X 0,Y 233.228,Z 660.777,A -85,B 0,C 180,E1 10771.305,E2 10771.305} C_VEL
LIN {X 0,Y 237.492,Z 672.472,A -85,B 0,C 180,E1 10766.818,E2 10766.818} C_VEL
LIN {X 0,Y 241.489,Z 684.517,A -85,B 0,C 180,E1 10762.808,E2 10762.808} C_VEL
LIN {X 0,Y 245.402,Z 697.614,A -85,B 0,C 180,E1 10759.046,E2 10759.046} C_VEL
LIN {X 0,Y 251.996,Z 711.241,A -85,B 0,C 180,E1 10757.41,E2 10757.41} C_VEL
LIN {X 0,Y 253.52,Z 739.011,A -85,B 0,C 180,E1 10756.194,E2 10756.194} C_VEL
LIN {X 0,Y 246.826,Z 878.333,A -85,B 0,C 180,E1 10752.479,E2 10752.479} C_VEL
LIN {X 0,Y 244.987,Z 896.523,A -85,B 0,C 180,E1 10751.613,E2 10751.613} C_VEL
LIN {X 0,Y 242.249,Z 914.072,A -85,B 0,C 180,E1 10750.392,E2 10750.392} C_VEL
LIN {X 0,Y 238.887,Z 931.273,A -85,B 0,C 180,E1 10748.737,E2 10748.737} C_VEL
LIN {X 0,Y 235.183,Z 947.384,A -85,B 0,C 180,E1 10746.679,E2 10746.679} C_VEL
LIN {X 0,Y 231.323,Z 962.516,A -85,B 0,C 180,E1 10744.189,E2 10744.189} C_VEL
LIN {X 0,Y 227.306,Z 977.205,A -85,B 0,C 180,E1 10741.122,E2 10741.122} C_VEL
LIN {X 0,Y 223.793,Z 990.224,A -85,B 0,C 180,E1 10737.688,E2 10737.688} C_VEL
LIN {X 0,Y 220.891,Z 1001.672,A -85,B 0,C 180,E1 10733.887,E2 10733.887} C_VEL
LIN {X 0,Y 218.784,Z 1011.61,A -85,B 0,C 180,E1 10729.707,E2 10729.707} C_VEL
LIN {X 0,Y 217.652,Z 1019.997,A -85,B 0,C 180,E1 10725.18,E2 10725.18} C_VEL
LIN {X 0,Y 217.525,Z 1026.395,A -85,B 0,C 180,E1 10720.595,E2 10720.595} C_VEL
LIN {X 0,Y 218.113,Z 1030.628,A -85,B 0,C 180,E1 10716.317,E2 10716.317} C_VEL
LIN {X 0,Y 218.795,Z 1033.053,A -85,B 0,C 180,E1 10712.358,E2 10712.358} C_VEL
LIN {X 0,Y 218.851,Z 1033.953,A -85,B 0,C 180,E1 10708.953,E2 10708.953} C_VEL
LIN {X 0,Y 218.174,Z 1033.62,A -85,B 0,C 180,E1 10705.269,E2 10705.269} C_VEL
LIN {X 0,Y 217.308,Z 1031.644,A -85,B 0,C 180,E1 10700.733,E2 10700.733} C_VEL
LIN {X 0,Y 217.194,Z 1027.791,A -85,B 0,C 180,E1 10695.878,E2 10695.878} C_VEL
LIN {X 0,Y 218.29,Z 1022.048,A -85,B 0,C 180,E1 10691.022,E2 10691.022} C_VEL
LIN {X 0,Y 220.829,Z 1014.29,A -85,B 0,C 180,E1 10686.236,E2 10686.236} C_VEL
LIN {X 0,Y 224.629,Z 1004.832,A -85,B 0,C 180,E1 10681.802,E2 10681.802} C_VEL
LIN {X 0,Y 229.339,Z 994.008,A -85,B 0,C 180,E1 10677.867,E2 10677.867} C_VEL
LIN {X 0,Y 234.512,Z 982.276,A -85,B 0,C 180,E1 10674.522,E2 10674.522} C_VEL
LIN {X 0,Y 239.991,Z 969.355,A -85,B 0,C 180,E1 10671.628,E2 10671.628} C_VEL
LIN {X 0,Y 245.696,Z 954.77,A -85,B 0,C 180,E1 10669.066,E2 10669.066} C_VEL
LIN {X 0,Y 251.174,Z 939.13,A -85,B 0,C 180,E1 10666.946,E2 10666.946} C_VEL
LIN {X 0,Y 255.961,Z 923.321,A -85,B 0,C 180,E1 10665.312,E2 10665.312} C_VEL
LIN {X 0,Y 260.25,Z 906.154,A -85,B 0,C 180,E1 10663.995,E2 10663.995} C_VEL
LIN {X 0,Y 263.525,Z 888.295,A -85,B 0,C 180,E1 10663.032,E2 10663.032} C_VEL
LIN {X 0,Y 265.579,Z 869.978,A -85,B 0,C 180,E1 10662.372,E2 10662.372} C_VEL
LIN {X 0,Y 273.889,Z 739.427,A -85,B 0,C 180,E1 10659.055,E2 10659.055} C_VEL
LIN {X 0,Y 273.396,Z 729.98,A -85,B 0,C 180,E1 10658.502,E2 10658.502} C_VEL
LIN {X 0,Y 267.191,Z 718.882,A -85,B 0,C 180,E1 10656.146,E2 10656.146} C_VEL
LIN {X 0,Y 260.647,Z 708.469,A -85,B 0,C 180,E1 10653.399,E2 10653.399} C_VEL
LIN {X 0,Y 256.636,Z 702.671,A -85,B 0,C 180,E1 10651.536,E2 10651.536} C_VEL
LIN {X 0,Y 254.057,Z 698.526,A -85,B 0,C 180,E1 10650.023,E2 10650.023} C_VEL
LIN {X 0,Y 251.749,Z 692.238,A -85,B 0,C 180,E1 10646.157,E2 10646.157} C_VEL
LIN {X 0,Y 249.686,Z 687.091,A -85,B 0,C 180,E1 10642.112,E2 10642.112} C_VEL
LIN {X 0,Y 248.277,Z 683.584,A -85,B 0,C 180,E1 10638.551,E2 10638.551} C_VEL
LIN {X 0,Y 246.713,Z 679.819,A -85,B 0,C 180,E1 10632.641,E2 10632.641} C_VEL
LIN {X 0,Y 245.815,Z 678.839,A -85,B 0,C 180,E1 10627.009,E2 10627.009} C_VEL
LIN {X 0,Y 246.121,Z 679.421,A -85,B 0,C 180,E1 10621.629,E2 10621.629} C_VEL
LIN {X 0,Y 247.013,Z 682.943,A -85,B 0,C 180,E1 10615.356,E2 10615.356} C_VEL
LIN {X 0,Y 248.019,Z 686.53,A -85,B 0,C 180,E1 10611.421,E2 10611.421} C_VEL
LIN {X 0,Y 249.106,Z 690.225,A -85,B 0,C 180,E1 10608.187,E2 10608.187} C_VEL
LIN {X 0,Y 250.74,Z 696.128,A -85,B 0,C 180,E1 10604.029,E2 10604.029} C_VEL
LIN {X 0,Y 252.429,Z 702.921,A -85,B 0,C 180,E1 10600.129,E2 10600.129} C_VEL
LIN {X 0,Y 257.546,Z 711.857,A -85,B 0,C 180,E1 10597.336,E2 10597.336} C_VEL
LIN {X 0,Y 261.827,Z 719.607,A -85,B 0,C 180,E1 10595.341,E2 10595.341} C_VEL
LIN {X 0,Y 265.446,Z 726.723,A -85,B 0,C 180,E1 10593.775,E2 10593.775} C_VEL
LIN {X 0,Y 269.018,Z 754.333,A -85,B 0,C 180,E1 10591.38,E2 10591.38} C_VEL
LIN {X 0,Y 270.011,Z 765.362,A -85,B 0,C 180,E1 10590.591,E2 10590.591} C_VEL
LIN {X 0,Y 264.267,Z 846.652,A -85,B 0,C 180,E1 10588.352,E2 10588.352} C_VEL
LIN {X 0,Y 262.35,Z 863.004,A -85,B 0,C 180,E1 10587.54,E2 10587.54} C_VEL
LIN {X 0,Y 259.443,Z 879.27,A -85,B 0,C 180,E1 10586.349,E2 10586.349} C_VEL
LIN {X 0,Y 255.973,Z 893.524,A -85,B 0,C 180,E1 10584.918,E2 10584.918} C_VEL
LIN {X 0,Y 251.596,Z 907.941,A -85,B 0,C 180,E1 10583.014,E2 10583.014} C_VEL
LIN {X 0,Y 246.978,Z 920.606,A -85,B 0,C 180,E1 10580.835,E2 10580.835} C_VEL
LIN {X 0,Y 241.786,Z 932.789,A -85,B 0,C 180,E1 10578.104,E2 10578.104} C_VEL
LIN {X 0,Y 236.927,Z 942.826,A -85,B 0,C 180,E1 10575.152,E2 10575.152} C_VEL
LIN {X 0,Y 232.286,Z 951.34,A -85,B 0,C 180,E1 10571.85,E2 10571.85} C_VEL
LIN {X 0,Y 228.079,Z 958.328,A -85,B 0,C 180,E1 10568.179,E2 10568.179} C_VEL
LIN {X 0,Y 224.433,Z 963.726,A -85,B 0,C 180,E1 10564.04,E2 10564.04} C_VEL
LIN {X 0,Y 221.903,Z 966.991,A -85,B 0,C 180,E1 10560.009,E2 10560.009} C_VEL
LIN {X 0,Y 220.125,Z 968.563,A -85,B 0,C 180,E1 10555.563,E2 10555.563} C_VEL
LIN {X 0,Y 219.295,Z 968.35,A -85,B 0,C 180,E1 10551.392,E2 10551.392} C_VEL
LIN {X 0,Y 219.163,Z 966.268,A -85,B 0,C 180,E1 10546.976,E2 10546.976} C_VEL
LIN {X 0,Y 219.729,Z 962.651,A -85,B 0,C 180,E1 10542.883,E2 10542.883} C_VEL
LIN {X 0,Y 220.996,Z 957.212,A -85,B 0,C 180,E1 10538.848,E2 10538.848} C_VEL
LIN {X 0,Y 223.028,Z 949.83,A -85,B 0,C 180,E1 10534.886,E2 10534.886} C_VEL
LIN {X 0,Y 225.425,Z 941.503,A -85,B 0,C 180,E1 10531.525,E2 10531.525} C_VEL
LIN {X 0,Y 228.406,Z 931.062,A -85,B 0,C 180,E1 10528.244,E2 10528.244} C_VEL
LIN {X 0,Y 231.484,Z 919.532,A -85,B 0,C 180,E1 10525.416,E2 10525.416} C_VEL
LIN {X 0,Y 234.65,Z 906.422,A -85,B 0,C 180,E1 10522.901,E2 10522.901} C_VEL
LIN {X 0,Y 237.479,Z 893.11,A -85,B 0,C 180,E1 10520.915,E2 10520.915} C_VEL
LIN {X 0,Y 240.09,Z 878.056,A -85,B 0,C 180,E1 10519.198,E2 10519.198} C_VEL
LIN {X 0,Y 242.172,Z 862.355,A -85,B 0,C 180,E1 10517.882,E2 10517.882} C_VEL
LIN {X 0,Y 243.688,Z 844.732,A -85,B 0,C 180,E1 10516.897,E2 10516.897} C_VEL
LIN {X 0,Y 247.364,Z 772.97,A -85,B 0,C 180,E1 10514.767,E2 10514.767} C_VEL
LIN {X 0,Y 248.034,Z 756.318,A -85,B 0,C 180,E1 10514.278,E2 10514.278} C_VEL
LIN {X 0,Y 241.383,Z 703.946,A -85,B 0,C 180,E1 10511.149,E2 10511.149} C_VEL
LIN {X 0,Y 242.125,Z 700.266,A -85,B 0,C 180,E1 10510.312,E2 10510.312} C_VEL
LIN {X 0,Y 239.332,Z 686.823,A -85,B 0,C 180,E1 10505.962,E2 10505.962} C_VEL
LIN {X 0,Y 236.29,Z 674.864,A -85,B 0,C 180,E1 10501.662,E2 10501.662} C_VEL
LIN {X 0,Y 233.048,Z 663.917,A -85,B 0,C 180,E1 10497.238,E2 10497.238} C_VEL
LIN {X 0,Y 229.696,Z 654.375,A -85,B 0,C 180,E1 10492.807,E2 10492.807} C_VEL
LIN {X 0,Y 226.843,Z 647.056,A -85,B 0,C 180,E1 10488.914,E2 10488.914} C_VEL
LIN {X 0,Y 224.305,Z 640.757,A -85,B 0,C 180,E1 10485.135,E2 10485.135} C_VEL
LIN {X 0,Y 222.507,Z 636.719,A -85,B 0,C 180,E1 10482.381,E2 10482.381} C_VEL
LIN {X 0,Y 220.536,Z 632.429,A -85,B 0,C 180,E1 10479.065,E2 10479.065} C_VEL
LIN {X 0,Y 218.906,Z 628.55,A -85,B 0,C 180,E1 10475.457,E2 10475.457} C_VEL
LIN {X 0,Y 218.889,Z 628.531,A -85,B 0,C 180,E1 10470.164,E2 10470.164} C_VEL
LIN {X 0,Y 218.895,Z 628.474,A -85,B 0,C 180,E1 10464.85,E2 10464.85} C_VEL
LIN {X 0,Y 218.882,Z 628.487,A -85,B 0,C 180,E1 10459.758,E2 10459.758} C_VEL
LIN {X 0,Y 218.908,Z 628.507,A -85,B 0,C 180,E1 10454.28,E2 10454.28} C_VEL
LIN {X 0,Y 218.881,Z 628.466,A -85,B 0,C 180,E1 10448.671,E2 10448.671} C_VEL
LIN {X 0,Y 218.882,Z 628.503,A -85,B 0,C 180,E1 10443.405,E2 10443.405} C_VEL
LIN {X 0,Y 218.887,Z 628.499,A -85,B 0,C 180,E1 10437.906,E2 10437.906} C_VEL
LIN {X 0,Y 218.869,Z 628.48,A -85,B 0,C 180,E1 10432.652,E2 10432.652} C_VEL
LIN {X 0,Y 218.943,Z 628.951,A -85,B 0,C 180,E1 10430.14,E2 10430.14} C_VEL
LIN {X 0,Y 219.196,Z 629.928,A -85,B 0,C 180,E1 10429.346,E2 10429.346} C_VEL
LIN {X 0,Y 219.399,Z 633.168,A -85,B 0,C 180,E1 10427.494,E2 10427.494} C_VEL
LIN {X 0,Y 218.415,Z 644.276,A -85,B 0,C 180,E1 10422.732,E2 10422.732} C_VEL
LIN {X 0,Y 219.28,Z 647.047,A -85,B 0,C 180,E1 10421.152,E2 10421.152} C_VEL
LIN {X 0,Y 222.161,Z 653.851,A -85,B 0,C 180,E1 10417.315,E2 10417.315} C_VEL
LIN {X 0,Y 225.747,Z 662.312,A -85,B 0,C 180,E1 10413.143,E2 10413.143} C_VEL
LIN {X 0,Y 229.606,Z 672.784,A -85,B 0,C 180,E1 10408.789,E2 10408.789} C_VEL
LIN {X 0,Y 233.698,Z 684.984,A -85,B 0,C 180,E1 10404.419,E2 10404.419} C_VEL
LIN {X 0,Y 237.513,Z 697.617,A -85,B 0,C 180,E1 10400.531,E2 10400.531} C_VEL
LIN {X 0,Y 245.63,Z 714.001,A -85,B 0,C 180,E1 10398.394,E2 10398.394} C_VEL
LIN {X 0,Y 246.958,Z 739.748,A -85,B 0,C 180,E1 10397.235,E2 10397.235} C_VEL
LIN {X 0,Y 240.065,Z 877.588,A -85,B 0,C 180,E1 10393.493,E2 10393.493} C_VEL
LIN {X 0,Y 238.167,Z 895.804,A -85,B 0,C 180,E1 10392.609,E2 10392.609} C_VEL
LIN {X 0,Y 235.319,Z 913.459,A -85,B 0,C 180,E1 10391.355,E2 10391.355} C_VEL
LIN {X 0,Y 231.839,Z 930.617,A -85,B 0,C 180,E1 10389.665,E2 10389.665} C_VEL
LIN {X 0,Y 227.999,Z 946.672,A -85,B 0,C 180,E1 10387.559,E2 10387.559} C_VEL
LIN {X 0,Y 223.986,Z 961.765,A -85,B 0,C 180,E1 10385.003,E2 10385.003} C_VEL
LIN {X 0,Y 219.806,Z 976.415,A -85,B 0,C 180,E1 10381.849,E2 10381.849} C_VEL
LIN {X 0,Y 216.26,Z 988.948,A -85,B 0,C 180,E1 10378.439,E2 10378.439} C_VEL
LIN {X 0,Y 213.192,Z 1000.433,A -85,B 0,C 180,E1 10374.516,E2 10374.516} C_VEL
LIN {X 0,Y 210.955,Z 1010.356,A -85,B 0,C 180,E1 10370.207,E2 10370.207} C_VEL
LIN {X 0,Y 209.724,Z 1018.808,A -85,B 0,C 180,E1 10365.485,E2 10365.485} C_VEL
LIN {X 0,Y 209.554,Z 1024.891,A -85,B 0,C 180,E1 10361.003,E2 10361.003} C_VEL
LIN {X 0,Y 210.135,Z 1029.236,A -85,B 0,C 180,E1 10356.558,E2 10356.558} C_VEL
LIN {X 0,Y 210.872,Z 1031.758,A -85,B 0,C 180,E1 10352.446,E2 10352.446} C_VEL
LIN {X 0,Y 210.969,Z 1032.697,A -85,B 0,C 180,E1 10349.186,E2 10349.186} C_VEL
LIN {X 0,Y 210.261,Z 1032.473,A -85,B 0,C 180,E1 10345.364,E2 10345.364} C_VEL
LIN {X 0,Y 209.342,Z 1030.648,A -85,B 0,C 180,E1 10340.655,E2 10340.655} C_VEL
LIN {X 0,Y 209.241,Z 1026.943,A -85,B 0,C 180,E1 10335.613,E2 10335.613} C_VEL
LIN {X 0,Y 210.425,Z 1021.395,A -85,B 0,C 180,E1 10330.573,E2 10330.573} C_VEL
LIN {X 0,Y 212.937,Z 1014.326,A -85,B 0,C 180,E1 10325.889,E2 10325.889} C_VEL
LIN {X 0,Y 216.825,Z 1005.27,A -85,B 0,C 180,E1 10321.342,E2 10321.342} C_VEL
LIN {X 0,Y 221.739,Z 994.691,A -85,B 0,C 180,E1 10317.242,E2 10317.242} C_VEL
LIN {X 0,Y 227.438,Z 982.568,A -85,B 0,C 180,E1 10313.596,E2 10313.596} C_VEL
LIN {X 0,Y 233.431,Z 969.316,A -85,B 0,C 180,E1 10310.501,E2 10310.501} C_VEL
LIN {X 0,Y 239.373,Z 954.93,A -85,B 0,C 180,E1 10307.902,E2 10307.902} C_VEL
LIN {X 0,Y 245.058,Z 939.527,A -85,B 0,C 180,E1 10305.758,E2 10305.758} C_VEL
LIN {X 0,Y 250.287,Z 923.079,A -85,B 0,C 180,E1 10304.022,E2 10304.022} C_VEL
LIN {X 0,Y 254.589,Z 906.727,A -85,B 0,C 180,E1 10302.743,E2 10302.743} C_VEL
LIN {X 0,Y 258.101,Z 888.972,A -85,B 0,C 180,E1 10301.747,E2 10301.747} C_VEL
LIN {X 0,Y 260.325,Z 870.776,A -85,B 0,C 180,E1 10301.066,E2 10301.066} C_VEL
LIN {X 0,Y 269.027,Z 740.396,A -85,B 0,C 180,E1 10297.72,E2 10297.72} C_VEL
LIN {X 0,Y 268.713,Z 734.127,A -85,B 0,C 180,E1 10297.337,E2 10297.337} C_VEL
LIN {X 0,Y 262.549,Z 722.928,A -85,B 0,C 180,E1 10294.836,E2 10294.836} C_VEL
LIN {X 0,Y 255.637,Z 711.831,A -85,B 0,C 180,E1 10291.673,E2 10291.673} C_VEL
LIN {X 0,Y 249.619,Z 703.479,A -85,B 0,C 180,E1 10288.532,E2 10288.532} C_VEL
LIN {X 0,Y 246.837,Z 699.315,A -85,B 0,C 180,E1 10286.719,E2 10286.719} C_VEL
LIN {X 0,Y 245.204,Z 695.284,A -85,B 0,C 180,E1 10283.809,E2 10283.809} C_VEL
LIN {X 0,Y 244.138,Z 692.515,A -85,B 0,C 180,E1 10281.376,E2 10281.376} C_VEL
LIN {X 0,Y 242.983,Z 689.504,A -85,B 0,C 180,E1 10278.224,E2 10278.224} C_VEL
LIN {X 0,Y 241.544,Z 685.911,A -85,B 0,C 180,E1 10272.43,E2 10272.43} C_VEL
LIN {X 0,Y 240.684,Z 684.967,A -85,B 0,C 180,E1 10266.679,E2 10266.679} C_VEL
LIN {X 0,Y 240.94,Z 685.54,A -85,B 0,C 180,E1 10261.664,E2 10261.664} C_VEL
LIN {X 0,Y 241.696,Z 688.934,A -85,B 0,C 180,E1 10255.476,E2 10255.476} C_VEL
LIN {X 0,Y 242.608,Z 692.513,A -85,B 0,C 180,E1 10251.467,E2 10251.467} C_VEL
LIN {X 0,Y 243.647,Z 696.231,A -85,B 0,C 180,E1 10248.159,E2 10248.159} C_VEL
LIN {X 0,Y 245.271,Z 702.389,A -85,B 0,C 180,E1 10243.784,E2 10243.784} C_VEL
LIN {X 0,Y 247.409,Z 706.474,A -85,B 0,C 180,E1 10242.112,E2 10242.112} C_VEL
LIN {X 0,Y 250.977,Z 712.274,A -85,B 0,C 180,E1 10240.024,E2 10240.024} C_VEL
LIN {X 0,Y 255.343,Z 719.824,A -85,B 0,C 180,E1 10237.737,E2 10237.737} C_VEL
LIN {X 0,Y 259.984,Z 728.525,A -85,B 0,C 180,E1 10235.519,E2 10235.519} C_VEL
LIN {X 0,Y 261.337,Z 731.903,A -85,B 0,C 180,E1 10234.869,E2 10234.869} C_VEL
LIN {X 0,Y 264.514,Z 758.923,A -85,B 0,C 180,E1 10232.492,E2 10232.492} C_VEL
LIN {X 0,Y 265.111,Z 766.906,A -85,B 0,C 180,E1 10231.927,E2 10231.927} C_VEL
LIN {X 0,Y 259.187,Z 847.461,A -85,B 0,C 180,E1 10229.694,E2 10229.694} C_VEL
LIN {X 0,Y 257.164,Z 863.878,A -85,B 0,C 180,E1 10228.87,E2 10228.87} C_VEL
LIN {X 0,Y 254.257,Z 879.506,A -85,B 0,C 180,E1 10227.723,E2 10227.723} C_VEL
LIN {X 0,Y 250.634,Z 893.943,A -85,B 0,C 180,E1 10226.281,E2 10226.281} C_VEL
LIN {X 0,Y 246.049,Z 908.439,A -85,B 0,C 180,E1 10224.363,E2 10224.363} C_VEL
LIN {X 0,Y 241.172,Z 921.255,A -85,B 0,C 180,E1 10222.15,E2 10222.15} C_VEL
LIN {X 0,Y 236.13,Z 932.557,A -85,B 0,C 180,E1 10219.619,E2 10219.619} C_VEL
LIN {X 0,Y 230.987,Z 942.796,A -85,B 0,C 180,E1 10216.653,E2 10216.653} C_VEL
LIN {X 0,Y 225.993,Z 951.555,A -85,B 0,C 180,E1 10213.295,E2 10213.295} C_VEL
LIN {X 0,Y 221.423,Z 958.781,A -85,B 0,C 180,E1 10209.546,E2 10209.546} C_VEL
LIN {X 0,Y 217.649,Z 964.108,A -85,B 0,C 180,E1 10205.597,E2 10205.597} C_VEL
LIN {X 0,Y 214.562,Z 967.889,A -85,B 0,C 180,E1 10201.148,E2 10201.148} C_VEL
LIN {X 0,Y 212.605,Z 969.653,A -85,B 0,C 180,E1 10196.838,E2 10196.838} C_VEL
LIN {X 0,Y 211.457,Z 969.633,A -85,B 0,C 180,E1 10192.061,E2 10192.061} C_VEL
LIN {X 0,Y 211.214,Z 967.84,A -85,B 0,C 180,E1 10187.636,E2 10187.636} C_VEL
LIN {X 0,Y 211.741,Z 964.133,A -85,B 0,C 180,E1 10183.1,E2 10183.1} C_VEL
LIN {X 0,Y 213.005,Z 958.86,A -85,B 0,C 180,E1 10178.911,E2 10178.911} C_VEL
LIN {X 0,Y 215.057,Z 951.608,A -85,B 0,C 180,E1 10174.8,E2 10174.8} C_VEL
LIN {X 0,Y 217.51,Z 943.512,A -85,B 0,C 180,E1 10171.317,E2 10171.317} C_VEL
LIN {X 0,Y 220.562,Z 933.267,A -85,B 0,C 180,E1 10167.921,E2 10167.921} C_VEL
LIN {X 0,Y 223.886,Z 921.523,A -85,B 0,C 180,E1 10164.875,E2 10164.875} C_VEL
LIN {X 0,Y 227.32,Z 907.938,A -85,B 0,C 180,E1 10162.163,E2 10162.163} C_VEL
LIN {X 0,Y 230.441,Z 893.923,A -85,B 0,C 180,E1 10160.005,E2 10160.005} C_VEL
LIN {X 0,Y 233.352,Z 877.73,A -85,B 0,C 180,E1 10158.131,E2 10158.131} C_VEL
LIN {X 0,Y 235.472,Z 861.924,A -85,B 0,C 180,E1 10156.814,E2 10156.814} C_VEL
LIN {X 0,Y 236.988,Z 844.698,A -85,B 0,C 180,E1 10155.851,E2 10155.851} C_VEL
LIN {X 0,Y 241.446,Z 757.326,A -85,B 0,C 180,E1 10153.222,E2 10153.222} C_VEL
LIN {X 0,Y 234.88,Z 703.772,A -85,B 0,C 180,E1 10149.894,E2 10149.894} C_VEL
LIN {X 0,Y 233.668,Z 696.378,A -85,B 0,C 180,E1 10147.558,E2 10147.558} C_VEL
LIN {X 0,Y 230.919,Z 684.083,A -85,B 0,C 180,E1 10143.236,E2 10143.236} C_VEL
LIN {X 0,Y 227.895,Z 672.892,A -85,B 0,C 180,E1 10138.82,E2 10138.82} C_VEL
LIN {X 0,Y 224.771,Z 662.925,A -85,B 0,C 180,E1 10134.356,E2 10134.356} C_VEL
LIN {X 0,Y 221.327,Z 653.357,A -85,B 0,C 180,E1 10129.373,E2 10129.373} C_VEL
LIN {X 0,Y 218.336,Z 645.993,A -85,B 0,C 180,E1 10124.85,E2 10124.85} C_VEL
LIN {X 0,Y 216.571,Z 641.962,A -85,B 0,C 180,E1 10121.985,E2 10121.985} C_VEL
LIN {X 0,Y 214.879,Z 638.064,A -85,B 0,C 180,E1 10118.916,E2 10118.916} C_VEL
LIN {X 0,Y 212.874,Z 633.778,A -85,B 0,C 180,E1 10114.962,E2 10114.962} C_VEL
LIN {X 0,Y 210.963,Z 629.609,A -85,B 0,C 180,E1 10109.845,E2 10109.845} C_VEL
LIN {X 0,Y 210.952,Z 629.466,A -85,B 0,C 180,E1 10104.488,E2 10104.488} C_VEL
LIN {X 0,Y 210.945,Z 629.464,A -85,B 0,C 180,E1 10099.091,E2 10099.091} C_VEL
LIN {X 0,Y 210.948,Z 629.513,A -85,B 0,C 180,E1 10093.668,E2 10093.668} C_VEL
LIN {X 0,Y 210.959,Z 629.453,A -85,B 0,C 180,E1 10088.175,E2 10088.175} C_VEL
LIN {X 0,Y 210.936,Z 629.476,A -85,B 0,C 180,E1 10082.717,E2 10082.717} C_VEL
LIN {X 0,Y 210.951,Z 629.503,A -85,B 0,C 180,E1 10077.556,E2 10077.556} C_VEL
LIN {X 0,Y 211.012,Z 629.911,A -85,B 0,C 180,E1 10075.653,E2 10075.653} C_VEL
LIN {X 0,Y 213.573,Z 635.167,A -85,B 0,C 180,E1 10070.026,E2 10070.026} C_VEL
LIN {X 0,Y 215.911,Z 639.879,A -85,B 0,C 180,E1 10066.066,E2 10066.066} C_VEL
LIN {X 0,Y 217.946,Z 644.327,A -85,B 0,C 180,E1 10062.926,E2 10062.926} C_VEL
LIN {X 0,Y 219.28,Z 647.047,A -85,B 0,C 180,E1 10061.152,E2 10061.152} C_VEL
LIN {X 0,Y 220.129,Z 649.947,A -85,B 0,C 180,E1 10059.619,E2 10059.619} C_VEL
LIN {X 0,Y 219.941,Z 655.075,A -85,B 0,C 180,E1 10057.722,E2 10057.722} C_VEL
LIN {X 0,Y 219.225,Z 664.89,A -85,B 0,C 180,E1 10054.47,E2 10054.47} C_VEL
LIN {X 0,Y 219.66,Z 667.353,A -85,B 0,C 180,E1 10053.484,E2 10053.484} C_VEL
LIN {X 0,Y 223.434,Z 677.833,A -85,B 0,C 180,E1 10049.028,E2 10049.028} C_VEL
LIN {X 0,Y 227.165,Z 689.364,A -85,B 0,C 180,E1 10044.789,E2 10044.789} C_VEL
LIN {X 0,Y 229.759,Z 697.906,A -85,B 0,C 180,E1 10042.071,E2 10042.071} C_VEL
LIN {X 0,Y 239.313,Z 716.832,A -85,B 0,C 180,E1 10039.423,E2 10039.423} C_VEL
LIN {X 0,Y 240.454,Z 740.508,A -85,B 0,C 180,E1 10038.324,E2 10038.324} C_VEL
LIN {X 0,Y 233.316,Z 877.122,A -85,B 0,C 180,E1 10034.538,E2 10034.538} C_VEL
LIN {X 0,Y 231.348,Z 895.345,A -85,B 0,C 180,E1 10033.632,E2 10033.632} C_VEL
LIN {X 0,Y 228.461,Z 912.68,A -85,B 0,C 180,E1 10032.376,E2 10032.376} C_VEL
LIN {X 0,Y 224.856,Z 929.857,A -85,B 0,C 180,E1 10030.651,E2 10030.651} C_VEL
LIN {X 0,Y 220.851,Z 945.988,A -85,B 0,C 180,E1 10028.484,E2 10028.484} C_VEL
LIN {X 0,Y 216.698,Z 960.999,A -85,B 0,C 180,E1 10025.873,E2 10025.873} C_VEL
LIN {X 0,Y 212.503,Z 975.09,A -85,B 0,C 180,E1 10022.759,E2 10022.759} C_VEL
LIN {X 0,Y 208.765,Z 987.671,A -85,B 0,C 180,E1 10019.244,E2 10019.244} C_VEL
LIN {X 0,Y 205.519,Z 999.196,A -85,B 0,C 180,E1 10015.191,E2 10015.191} C_VEL
LIN {X 0,Y 203.142,Z 1009.102,A -85,B 0,C 180,E1 10010.744,E2 10010.744} C_VEL
LIN {X 0,Y 201.834,Z 1017.268,A -85,B 0,C 180,E1 10006.045,E2 10006.045} C_VEL
LIN {X 0,Y 201.6,Z 1023.711,A -85,B 0,C 180,E1 10001.153,E2 10001.153} C_VEL
LIN {X 0,Y 202.228,Z 1028.166,A -85,B 0,C 180,E1 9996.394,E2 9996.394} C_VEL
LIN {X 0,Y 202.985,Z 1030.574,A -85,B 0,C 180,E1 9992.259,E2 9992.259} C_VEL
LIN {X 0,Y 203.025,Z 1031.485,A -85,B 0,C 180,E1 9988.872,E2 9988.872} C_VEL
LIN {X 0,Y 202.213,Z 1031.216,A -85,B 0,C 180,E1 9984.894,E2 9984.894} C_VEL
LIN {X 0,Y 201.308,Z 1029.344,A -85,B 0,C 180,E1 9979.989,E2 9979.989} C_VEL
LIN {X 0,Y 201.36,Z 1025.6,A -85,B 0,C 180,E1 9974.742,E2 9974.742} C_VEL
LIN {X 0,Y 202.823,Z 1019.995,A -85,B 0,C 180,E1 9969.495,E2 9969.495} C_VEL
LIN {X 0,Y 205.873,Z 1012.419,A -85,B 0,C 180,E1 9964.39,E2 9964.39} C_VEL
LIN {X 0,Y 210.239,Z 1003.213,A -85,B 0,C 180,E1 9959.728,E2 9959.728} C_VEL
LIN {X 0,Y 215.63,Z 992.449,A -85,B 0,C 180,E1 9955.549,E2 9955.549} C_VEL
LIN {X 0,Y 221.357,Z 980.985,A -85,B 0,C 180,E1 9952.099,E2 9952.099} C_VEL
LIN {X 0,Y 227.706,Z 967.594,A -85,B 0,C 180,E1 9948.97,E2 9948.97} C_VEL
LIN {X 0,Y 234.03,Z 952.946,A -85,B 0,C 180,E1 9946.333,E2 9946.333} C_VEL
LIN {X 0,Y 239.932,Z 937.565,A -85,B 0,C 180,E1 9944.212,E2 9944.212} C_VEL
LIN {X 0,Y 245.085,Z 921.93,A -85,B 0,C 180,E1 9942.577,E2 9942.577} C_VEL
LIN {X 0,Y 249.714,Z 904.847,A -85,B 0,C 180,E1 9941.258,E2 9941.258} C_VEL
LIN {X 0,Y 253.231,Z 887.073,A -85,B 0,C 180,E1 9940.29,E2 9940.29} C_VEL
LIN {X 0,Y 255.447,Z 868.953,A -85,B 0,C 180,E1 9939.628,E2 9939.628} C_VEL
LIN {X 0,Y 264.32,Z 741.51,A -85,B 0,C 180,E1 9936.344,E2 9936.344} C_VEL
LIN {X 0,Y 264.078,Z 738.124,A -85,B 0,C 180,E1 9936.102,E2 9936.102} C_VEL
LIN {X 0,Y 258.013,Z 727.169,A -85,B 0,C 180,E1 9933.452,E2 9933.452} C_VEL
LIN {X 0,Y 252.426,Z 718.053,A -85,B 0,C 180,E1 9930.728,E2 9930.728} C_VEL
LIN {X 0,Y 247.317,Z 710.636,A -85,B 0,C 180,E1 9927.901,E2 9927.901} C_VEL
LIN {X 0,Y 243.249,Z 704.963,A -85,B 0,C 180,E1 9925.308,E2 9925.308} C_VEL
LIN {X 0,Y 239.366,Z 699.414,A -85,B 0,C 180,E1 9922.147,E2 9922.147} C_VEL
LIN {X 0,Y 237.801,Z 695.586,A -85,B 0,C 180,E1 9918.128,E2 9918.128} C_VEL
LIN {X 0,Y 236.399,Z 692.028,A -85,B 0,C 180,E1 9912.306,E2 9912.306} C_VEL
LIN {X 0,Y 235.552,Z 691.104,A -85,B 0,C 180,E1 9906.581,E2 9906.581} C_VEL
LIN {X 0,Y 235.749,Z 691.658,A -85,B 0,C 180,E1 9901.701,E2 9901.701} C_VEL
LIN {X 0,Y 236.387,Z 694.904,A -85,B 0,C 180,E1 9895.633,E2 9895.633} C_VEL
LIN {X 0,Y 237.208,Z 698.495,A -85,B 0,C 180,E1 9891.516,E2 9891.516} C_VEL
LIN {X 0,Y 238.195,Z 702.182,A -85,B 0,C 180,E1 9888.191,E2 9888.191} C_VEL
LIN {X 0,Y 240.9,Z 706.935,A -85,B 0,C 180,E1 9885.702,E2 9885.702} C_VEL
LIN {X 0,Y 243.995,Z 711.71,A -85,B 0,C 180,E1 9883.52,E2 9883.52} C_VEL
LIN {X 0,Y 248.169,Z 718.744,A -85,B 0,C 180,E1 9880.891,E2 9880.891} C_VEL
LIN {X 0,Y 252.456,Z 726.472,A -85,B 0,C 180,E1 9878.509,E2 9878.509} C_VEL
LIN {X 0,Y 257.049,Z 735.57,A -85,B 0,C 180,E1 9876.198,E2 9876.198} C_VEL
LIN {X 0,Y 258.864,Z 750.712,A -85,B 0,C 180,E1 9874.735,E2 9874.735} C_VEL
LIN {X 0,Y 260.388,Z 768.109,A -85,B 0,C 180,E1 9873.32,E2 9873.32} C_VEL
LIN {X 0,Y 254.274,Z 848.012,A -85,B 0,C 180,E1 9871.098,E2 9871.098} C_VEL
LIN {X 0,Y 252.182,Z 864.396,A -85,B 0,C 180,E1 9870.276,E2 9870.276} C_VEL
LIN {X 0,Y 249.016,Z 880.707,A -85,B 0,C 180,E1 9869.072,E2 9869.072} C_VEL
LIN {X 0,Y 245.153,Z 895.303,A -85,B 0,C 180,E1 9867.591,E2 9867.591} C_VEL
LIN {X 0,Y 240.289,Z 909.946,A -85,B 0,C 180,E1 9865.623,E2 9865.623} C_VEL
LIN {X 0,Y 235.291,Z 922.411,A -85,B 0,C 180,E1 9863.431,E2 9863.431} C_VEL
LIN {X 0,Y 229.57,Z 934.562,A -85,B 0,C 180,E1 9860.641,E2 9860.641} C_VEL
LIN {X 0,Y 224.334,Z 944.367,A -85,B 0,C 180,E1 9857.699,E2 9857.699} C_VEL
LIN {X 0,Y 218.993,Z 953.132,A -85,B 0,C 180,E1 9854.207,E2 9854.207} C_VEL
LIN {X 0,Y 214.271,Z 960.121,A -85,B 0,C 180,E1 9850.437,E2 9850.437} C_VEL
LIN {X 0,Y 210.331,Z 965.302,A -85,B 0,C 180,E1 9846.456,E2 9846.456} C_VEL
LIN {X 0,Y 206.955,Z 969.14,A -85,B 0,C 180,E1 9841.776,E2 9841.776} C_VEL
LIN {X 0,Y 204.839,Z 970.879,A -85,B 0,C 180,E1 9837.311,E2 9837.311} C_VEL
LIN {X 0,Y 203.603,Z 970.87,A -85,B 0,C 180,E1 9832.522,E2 9832.522} C_VEL
LIN {X 0,Y 203.284,Z 969.223,A -85,B 0,C 180,E1 9828.051,E2 9828.051} C_VEL
LIN {X 0,Y 203.755,Z 965.61,A -85,B 0,C 180,E1 9823.334,E2 9823.334} C_VEL
LIN {X 0,Y 205.01,Z 960.485,A -85,B 0,C 180,E1 9818.978,E2 9818.978} C_VEL
LIN {X 0,Y 207.085,Z 953.371,A -85,B 0,C 180,E1 9814.708,E2 9814.708} C_VEL
LIN {X 0,Y 209.81,Z 944.761,A -85,B 0,C 180,E1 9810.819,E2 9810.819} C_VEL
LIN {X 0,Y 212.99,Z 934.564,A -85,B 0,C 180,E1 9807.309,E2 9807.309} C_VEL
LIN {X 0,Y 216.454,Z 922.889,A -85,B 0,C 180,E1 9804.167,E2 9804.167} C_VEL
LIN {X 0,Y 219.856,Z 910.092,A -85,B 0,C 180,E1 9801.5,E2 9801.5} C_VEL
LIN {X 0,Y 223.274,Z 895.581,A -85,B 0,C 180,E1 9799.159,E2 9799.159} C_VEL
LIN {X 0,Y 226.108,Z 880.739,A -85,B 0,C 180,E1 9797.356,E2 9797.356} C_VEL
LIN {X 0,Y 228.437,Z 865.042,A -85,B 0,C 180,E1 9795.94,E2 9795.94} C_VEL
LIN {X 0,Y 230.087,Z 848.221,A -85,B 0,C 180,E1 9794.918,E2 9794.918} C_VEL
LIN {X 0,Y 231.616,Z 820.468,A -85,B 0,C 180,E1 9793.957,E2 9793.957} C_VEL
LIN {X 0,Y 234.952,Z 758.462,A -85,B 0,C 180,E1 9792.117,E2 9792.117} C_VEL
LIN {X 0,Y 228.662,Z 706.636,A -85,B 0,C 180,E1 9788.824,E2 9788.824} C_VEL
LIN {X 0,Y 227.416,Z 703.529,A -85,B 0,C 180,E1 9788.326,E2 9788.326} C_VEL
LIN {X 0,Y 224.834,Z 690.987,A -85,B 0,C 180,E1 9783.939,E2 9783.939} C_VEL
LIN {X 0,Y 222.066,Z 679.882,A -85,B 0,C 180,E1 9779.566,E2 9779.566} C_VEL
LIN {X 0,Y 219.216,Z 670.022,A -85,B 0,C 180,E1 9775.185,E2 9775.185} C_VEL
LIN {X 0,Y 216.156,Z 661.08,A -85,B 0,C 180,E1 9770.578,E2 9770.578} C_VEL
LIN {X 0,Y 213.541,Z 654.236,A -85,B 0,C 180,E1 9766.504,E2 9766.504} C_VEL
LIN {X 0,Y 211.874,Z 650.219,A -85,B 0,C 180,E1 9763.777,E2 9763.777} C_VEL
LIN {X 0,Y 210.693,Z 647.271,A -85,B 0,C 180,E1 9761.636,E2 9761.636} C_VEL
LIN {X 0,Y 209.005,Z 643.408,A -85,B 0,C 180,E1 9758.456,E2 9758.456} C_VEL
LIN {X 0,Y 207.263,Z 639.435,A -85,B 0,C 180,E1 9754.698,E2 9754.698} C_VEL
LIN {X 0,Y 205.074,Z 634.94,A -85,B 0,C 180,E1 9749.181,E2 9749.181} C_VEL
LIN {X 0,Y 203.053,Z 630.699,A -85,B 0,C 180,E1 9740.675,E2 9740.675} C_VEL
LIN {X 0,Y 203.004,Z 630.465,A -85,B 0,C 180,E1 9735.121,E2 9735.121} C_VEL
LIN {X 0,Y 203.005,Z 630.474,A -85,B 0,C 180,E1 9729.641,E2 9729.641} C_VEL
LIN {X 0,Y 203.053,Z 630.838,A -85,B 0,C 180,E1 9725.086,E2 9725.086} C_VEL
LIN {X 0,Y 205.623,Z 635.61,A -85,B 0,C 180,E1 9716.097,E2 9716.097} C_VEL
LIN {X 0,Y 208.126,Z 640.933,A -85,B 0,C 180,E1 9710.321,E2 9710.321} C_VEL
LIN {X 0,Y 210.278,Z 645.3,A -85,B 0,C 180,E1 9706.527,E2 9706.527} C_VEL
LIN {X 0,Y 212.384,Z 650.191,A -85,B 0,C 180,E1 9703.03,E2 9703.03} C_VEL
LIN {X 0,Y 214.269,Z 654.341,A -85,B 0,C 180,E1 9700.368,E2 9700.368} C_VEL
LIN {X 0,Y 217.272,Z 661.446,A -85,B 0,C 180,E1 9696.4,E2 9696.4} C_VEL
LIN {X 0,Y 219.66,Z 667.353,A -85,B 0,C 180,E1 9693.484,E2 9693.484} C_VEL
LIN {X 0,Y 220.168,Z 671.889,A -85,B 0,C 180,E1 9691.842,E2 9691.842} C_VEL
LIN {X 0,Y 219.007,Z 687.059,A -85,B 0,C 180,E1 9687.52,E2 9687.52} C_VEL
LIN {X 0,Y 219.639,Z 690.431,A -85,B 0,C 180,E1 9686.368,E2 9686.368} C_VEL
LIN {X 0,Y 222.012,Z 698.116,A -85,B 0,C 180,E1 9683.765,E2 9683.765} C_VEL
LIN {X 0,Y 231.499,Z 716.509,A -85,B 0,C 180,E1 9680.947,E2 9680.947} C_VEL
LIN {X 0,Y 233.131,Z 720.333,A -85,B 0,C 180,E1 9680.47,E2 9680.47} C_VEL
LIN {X 0,Y 234.035,Z 741.367,A -85,B 0,C 180,E1 9679.471,E2 9679.471} C_VEL
LIN {X 0,Y 226.658,Z 876.538,A -85,B 0,C 180,E1 9675.648,E2 9675.648} C_VEL
LIN {X 0,Y 224.611,Z 894.818,A -85,B 0,C 180,E1 9674.719,E2 9674.719} C_VEL
LIN {X 0,Y 221.528,Z 912.626,A -85,B 0,C 180,E1 9673.393,E2 9673.393} C_VEL
LIN {X 0,Y 217.944,Z 929.024,A -85,B 0,C 180,E1 9671.7,E2 9671.7} C_VEL
LIN {X 0,Y 213.809,Z 945.069,A -85,B 0,C 180,E1 9669.495,E2 9669.495} C_VEL
LIN {X 0,Y 209.466,Z 960.143,A -85,B 0,C 180,E1 9666.803,E2 9666.803} C_VEL
LIN {X 0,Y 205.092,Z 974.227,A -85,B 0,C 180,E1 9663.597,E2 9663.597} C_VEL
LIN {X 0,Y 201.044,Z 987.254,A -85,B 0,C 180,E1 9659.825,E2 9659.825} C_VEL
LIN {X 0,Y 197.775,Z 998.294,A -85,B 0,C 180,E1 9655.772,E2 9655.772} C_VEL
LIN {X 0,Y 195.339,Z 1007.874,A -85,B 0,C 180,E1 9651.311,E2 9651.311} C_VEL
LIN {X 0,Y 193.926,Z 1015.995,A -85,B 0,C 180,E1 9646.466,E2 9646.466} C_VEL
LIN {X 0,Y 193.645,Z 1022.529,A -85,B 0,C 180,E1 9641.316,E2 9641.316} C_VEL
LIN {X 0,Y 194.27,Z 1026.879,A -85,B 0,C 180,E1 9636.502,E2 9636.502} C_VEL
LIN {X 0,Y 195.059,Z 1029.272,A -85,B 0,C 180,E1 9632.351,E2 9632.351} C_VEL
LIN {X 0,Y 195.155,Z 1030.176,A -85,B 0,C 180,E1 9629.12,E2 9629.12} C_VEL
LIN {X 0,Y 194.296,Z 1030.069,A -85,B 0,C 180,E1 9624.982,E2 9624.982} C_VEL
LIN {X 0,Y 193.341,Z 1028.347,A -85,B 0,C 180,E1 9619.874,E2 9619.874} C_VEL
LIN {X 0,Y 193.47,Z 1024.512,A -85,B 0,C 180,E1 9614.104,E2 9614.104} C_VEL
LIN {X 0,Y 195.135,Z 1019.003,A -85,B 0,C 180,E1 9608.667,E2 9608.667} C_VEL
LIN {X 0,Y 198.254,Z 1011.994,A -85,B 0,C 180,E1 9603.653,E2 9603.653} C_VEL
LIN {X 0,Y 202.867,Z 1002.974,A -85,B 0,C 180,E1 9598.835,E2 9598.835} C_VEL
LIN {X 0,Y 208.528,Z 992.401,A -85,B 0,C 180,E1 9594.537,E2 9594.537} C_VEL
LIN {X 0,Y 214.975,Z 980.304,A -85,B 0,C 180,E1 9590.762,E2 9590.762} C_VEL
LIN {X 0,Y 221.642,Z 967.075,A -85,B 0,C 180,E1 9587.591,E2 9587.591} C_VEL
LIN {X 0,Y 228.182,Z 952.695,A -85,B 0,C 180,E1 9584.955,E2 9584.955} C_VEL
LIN {X 0,Y 234.384,Z 937.28,A -85,B 0,C 180,E1 9582.8,E2 9582.8} C_VEL
LIN {X 0,Y 240.05,Z 920.781,A -85,B 0,C 180,E1 9581.071,E2 9581.071} C_VEL
LIN {X 0,Y 244.844,Z 903.587,A -85,B 0,C 180,E1 9579.759,E2 9579.759} C_VEL
LIN {X 0,Y 248.451,Z 885.697,A -85,B 0,C 180,E1 9578.8,E2 9578.8} C_VEL
LIN {X 0,Y 250.745,Z 867.058,A -85,B 0,C 180,E1 9578.132,E2 9578.132} C_VEL
LIN {X 0,Y 259.797,Z 742.698,A -85,B 0,C 180,E1 9574.916,E2 9574.916} C_VEL
LIN {X 0,Y 254.581,Z 733.029,A -85,B 0,C 180,E1 9572.485,E2 9572.485} C_VEL
LIN {X 0,Y 249.296,Z 724.237,A -85,B 0,C 180,E1 9569.757,E2 9569.757} C_VEL
LIN {X 0,Y 244.858,Z 717.536,A -85,B 0,C 180,E1 9567.143,E2 9567.143} C_VEL
LIN {X 0,Y 240.946,Z 711.903,A -85,B 0,C 180,E1 9564.517,E2 9564.517} C_VEL
LIN {X 0,Y 236.911,Z 706.468,A -85,B 0,C 180,E1 9561.281,E2 9561.281} C_VEL
LIN {X 0,Y 233.102,Z 701.869,A -85,B 0,C 180,E1 9557.472,E2 9557.472} C_VEL
LIN {X 0,Y 231.608,Z 699.414,A -85,B 0,C 180,E1 9554.5,E2 9554.5} C_VEL
LIN {X 0,Y 231.204,Z 698.098,A -85,B 0,C 180,E1 9551.98,E2 9551.98} C_VEL
LIN {X 0,Y 230.422,Z 697.253,A -85,B 0,C 180,E1 9546.227,E2 9546.227} C_VEL
LIN {X 0,Y 230.58,Z 697.799,A -85,B 0,C 180,E1 9541.739,E2 9541.739} C_VEL
LIN {X 0,Y 231.083,Z 700.887,A -85,B 0,C 180,E1 9535.781,E2 9535.781} C_VEL
LIN {X 0,Y 232.071,Z 703.363,A -85,B 0,C 180,E1 9533.195,E2 9533.195} C_VEL
LIN {X 0,Y 236.904,Z 710.755,A -85,B 0,C 180,E1 9528.064,E2 9528.064} C_VEL
LIN {X 0,Y 241.518,Z 718.38,A -85,B 0,C 180,E1 9524.389,E2 9524.389} C_VEL
LIN {X 0,Y 245.516,Z 725.385,A -85,B 0,C 180,E1 9521.724,E2 9521.724} C_VEL
LIN {X 0,Y 249.617,Z 733.119,A -85,B 0,C 180,E1 9519.298,E2 9519.298} C_VEL
LIN {X 0,Y 253.335,Z 740.912,A -85,B 0,C 180,E1 9517.306,E2 9517.306} C_VEL
LIN {X 0,Y 255.796,Z 767.386,A -85,B 0,C 180,E1 9514.905,E2 9514.905} C_VEL
LIN {X 0,Y 255.732,Z 771.145,A -85,B 0,C 180,E1 9514.724,E2 9514.724} C_VEL
LIN {X 0,Y 249.533,Z 848.713,A -85,B 0,C 180,E1 9512.555,E2 9512.555} C_VEL
LIN {X 0,Y 247.345,Z 865.085,A -85,B 0,C 180,E1 9511.73,E2 9511.73} C_VEL
LIN {X 0,Y 244.15,Z 880.894,A -85,B 0,C 180,E1 9510.565,E2 9510.565} C_VEL
LIN {X 0,Y 240.109,Z 895.722,A -85,B 0,C 180,E1 9509.073,E2 9509.073} C_VEL
LIN {X 0,Y 235.026,Z 910.443,A -85,B 0,C 180,E1 9507.097,E2 9507.097} C_VEL
LIN {X 0,Y 229.788,Z 923.032,A -85,B 0,C 180,E1 9504.888,E2 9504.888} C_VEL
LIN {X 0,Y 224.006,Z 934.795,A -85,B 0,C 180,E1 9502.189,E2 9502.189} C_VEL
LIN {X 0,Y 218.174,Z 945.234,A -85,B 0,C 180,E1 9499.053,E2 9499.053} C_VEL
LIN {X 0,Y 212.495,Z 954.081,A -85,B 0,C 180,E1 9495.484,E2 9495.484} C_VEL
LIN {X 0,Y 207.511,Z 961.034,A -85,B 0,C 180,E1 9491.677,E2 9491.677} C_VEL
LIN {X 0,Y 203.26,Z 966.309,A -85,B 0,C 180,E1 9487.587,E2 9487.587} C_VEL
LIN {X 0,Y 199.756,Z 970.022,A -85,B 0,C 180,E1 9483.065,E2 9483.065} C_VEL
LIN {X 0,Y 197.333,Z 971.983,A -85,B 0,C 180,E1 9478.443,E2 9478.443} C_VEL
LIN {X 0,Y 195.909,Z 972.23,A -85,B 0,C 180,E1 9473.777,E2 9473.777} C_VEL
LIN {X 0,Y 195.36,Z 970.694,A -85,B 0,C 180,E1 9468.764,E2 9468.764} C_VEL
LIN {X 0,Y 195.675,Z 967.651,A -85,B 0,C 180,E1 9464.197,E2 9464.197} C_VEL
LIN {X 0,Y 196.899,Z 962.449,A -85,B 0,C 180,E1 9459.351,E2 9459.351} C_VEL
LIN {X 0,Y 198.948,Z 955.677,A -85,B 0,C 180,E1 9454.901,E2 9454.901} C_VEL
LIN {X 0,Y 201.67,Z 947.339,A -85,B 0,C 180,E1 9450.852,E2 9450.852} C_VEL
LIN {X 0,Y 204.896,Z 937.605,A -85,B 0,C 180,E1 9447.202,E2 9447.202} C_VEL
LIN {X 0,Y 208.525,Z 925.982,A -85,B 0,C 180,E1 9443.851,E2 9443.851} C_VEL
LIN {X 0,Y 212.074,Z 913.585,A -85,B 0,C 180,E1 9441.049,E2 9441.049} C_VEL
LIN {X 0,Y 215.553,Z 899.767,A -85,B 0,C 180,E1 9438.646,E2 9438.646} C_VEL
LIN {X 0,Y 218.714,Z 884.828,A -85,B 0,C 180,E1 9436.652,E2 9436.652} C_VEL
LIN {X 0,Y 221.233,Z 869.438,A -85,B 0,C 180,E1 9435.138,E2 9435.138} C_VEL
LIN {X 0,Y 223.202,Z 852.433,A -85,B 0,C 180,E1 9433.966,E2 9433.966} C_VEL
LIN {X 0,Y 224.41,Z 832.956,A -85,B 0,C 180,E1 9433.177,E2 9433.177} C_VEL
LIN {X 0,Y 228.53,Z 759.421,A -85,B 0,C 180,E1 9430.939,E2 9430.939} C_VEL
LIN {X 0,Y 222.741,Z 709.921,A -85,B 0,C 180,E1 9427.673,E2 9427.673} C_VEL
LIN {X 0,Y 219.765,Z 703.367,A -85,B 0,C 180,E1 9426.611,E2 9426.611} C_VEL
LIN {X 0,Y 217.236,Z 691.224,A -85,B 0,C 180,E1 9422.094,E2 9422.094} C_VEL
LIN {X 0,Y 214.492,Z 680.471,A -85,B 0,C 180,E1 9417.538,E2 9417.538} C_VEL
LIN {X 0,Y 211.767,Z 671.381,A -85,B 0,C 180,E1 9413.156,E2 9413.156} C_VEL
LIN {X 0,Y 209.058,Z 663.32,A -85,B 0,C 180,E1 9408.668,E2 9408.668} C_VEL
LIN {X 0,Y 206.448,Z 656.48,A -85,B 0,C 180,E1 9404.209,E2 9404.209} C_VEL
LIN {X 0,Y 204.818,Z 652.551,A -85,B 0,C 180,E1 9401.227,E2 9401.227} C_VEL
LIN {X 0,Y 203.364,Z 649.047,A -85,B 0,C 180,E1 9398.28,E2 9398.28} C_VEL
LIN {X 0,Y 201.66,Z 645.1,A -85,B 0,C 180,E1 9394.419,E2 9394.419} C_VEL
LIN {X 0,Y 199.693,Z 640.846,A -85,B 0,C 180,E1 9389.058,E2 9389.058} C_VEL
LIN {X 0,Y 197.687,Z 636.6,A -85,B 0,C 180,E1 9380.426,E2 9380.426} C_VEL
LIN {X 0,Y 196.995,Z 635.74,A -85,B 0,C 180,E1 9374.2,E2 9374.2} C_VEL
LIN {X 0,Y 197.378,Z 636.182,A -85,B 0,C 180,E1 9367.862,E2 9367.862} C_VEL
LIN {X 0,Y 197.968,Z 637.394,A -85,B 0,C 180,E1 9364.055,E2 9364.055} C_VEL
LIN {X 0,Y 200.378,Z 641.877,A -85,B 0,C 180,E1 9355.995,E2 9355.995} C_VEL
LIN {X 0,Y 202.665,Z 646.682,A -85,B 0,C 180,E1 9350.631,E2 9350.631} C_VEL
LIN {X 0,Y 204.756,Z 651.107,A -85,B 0,C 180,E1 9346.732,E2 9346.732} C_VEL
LIN {X 0,Y 206.836,Z 656.035,A -85,B 0,C 180,E1 9343.14,E2 9343.14} C_VEL
LIN {X 0,Y 208.674,Z 660.237,A -85,B 0,C 180,E1 9340.403,E2 9340.403} C_VEL
LIN {X 0,Y 211.638,Z 667.458,A -85,B 0,C 180,E1 9336.324,E2 9336.324} C_VEL
LIN {X 0,Y 215.042,Z 676.433,A -85,B 0,C 180,E1 9331.992,E2 9331.992} C_VEL
LIN {X 0,Y 218.817,Z 687.735,A -85,B 0,C 180,E1 9327.372,E2 9327.372} C_VEL
LIN {X 0,Y 219.639,Z 690.431,A -85,B 0,C 180,E1 9326.368,E2 9326.368} C_VEL
LIN {X 0,Y 220.724,Z 694.946,A -85,B 0,C 180,E1 9325.147,E2 9325.147} C_VEL
LIN {X 0,Y 221.835,Z 702.477,A -85,B 0,C 180,E1 9323.953,E2 9323.953} C_VEL
LIN {X 0,Y 224.275,Z 715.951,A -85,B 0,C 180,E1 9322.5,E2 9322.5} C_VEL
LIN {X 0,Y 226.003,Z 720.864,A -85,B 0,C 180,E1 9321.912,E2 9321.912} C_VEL
LIN {X 0,Y 227.004,Z 723.599,A -85,B 0,C 180,E1 9321.588,E2 9321.588} C_VEL
LIN {X 0,Y 227.717,Z 742.205,A -85,B 0,C 180,E1 9320.682,E2 9320.682} C_VEL
LIN {X 0,Y 220.092,Z 875.916,A -85,B 0,C 180,E1 9316.827,E2 9316.827} C_VEL
LIN {X 0,Y 217.976,Z 894.171,A -85,B 0,C 180,E1 9315.88,E2 9315.88} C_VEL
LIN {X 0,Y 214.849,Z 911.674,A -85,B 0,C 180,E1 9314.553,E2 9314.553} C_VEL
LIN {X 0,Y 211.084,Z 928.295,A -85,B 0,C 180,E1 9312.805,E2 9312.805} C_VEL
LIN {X 0,Y 206.815,Z 944.228,A -85,B 0,C 180,E1 9310.561,E2 9310.561} C_VEL
LIN {X 0,Y 202.292,Z 959.285,A -85,B 0,C 180,E1 9307.8,E2 9307.8} C_VEL
LIN {X 0,Y 197.709,Z 973.414,A -85,B 0,C 180,E1 9304.48,E2 9304.48} C_VEL
LIN {X 0,Y 193.625,Z 985.902,A -85,B 0,C 180,E1 9300.746,E2 9300.746} C_VEL
LIN {X 0,Y 190.158,Z 997.007,A -85,B 0,C 180,E1 9296.548,E2 9296.548} C_VEL
LIN {X 0,Y 187.554,Z 1006.631,A -85,B 0,C 180,E1 9291.912,E2 9291.912} C_VEL
LIN {X 0,Y 186.02,Z 1014.775,A -85,B 0,C 180,E1 9286.874,E2 9286.874} C_VEL
LIN {X 0,Y 185.689,Z 1021.354,A -85,B 0,C 180,E1 9281.482,E2 9281.482} C_VEL
LIN {X 0,Y 186.336,Z 1025.7,A -85,B 0,C 180,E1 9276.471,E2 9276.471} C_VEL
LIN {X 0,Y 187.174,Z 1028.085,A -85,B 0,C 180,E1 9272.144,E2 9272.144} C_VEL
LIN {X 0,Y 187.246,Z 1028.916,A -85,B 0,C 180,E1 9269.083,E2 9269.083} C_VEL
LIN {X 0,Y 186.378,Z 1028.922,A -85,B 0,C 180,E1 9265.077,E2 9265.077} C_VEL
LIN {X 0,Y 185.372,Z 1027.357,A -85,B 0,C 180,E1 9259.748,E2 9259.748} C_VEL
LIN {X 0,Y 185.493,Z 1023.93,A -85,B 0,C 180,E1 9254.044,E2 9254.044} C_VEL
LIN {X 0,Y 187.347,Z 1018.335,A -85,B 0,C 180,E1 9248.064,E2 9248.064} C_VEL
LIN {X 0,Y 190.913,Z 1011.053,A -85,B 0,C 180,E1 9242.557,E2 9242.557} C_VEL
LIN {X 0,Y 195.882,Z 1002.136,A -85,B 0,C 180,E1 9237.591,E2 9237.591} C_VEL
LIN {X 0,Y 201.912,Z 991.672,A -85,B 0,C 180,E1 9233.189,E2 9233.189} C_VEL
LIN {X 0,Y 208.722,Z 979.668,A -85,B 0,C 180,E1 9229.346,E2 9229.346} C_VEL
LIN {X 0,Y 215.712,Z 966.539,A -85,B 0,C 180,E1 9226.136,E2 9226.136} C_VEL
LIN {X 0,Y 222.542,Z 952.292,A -85,B 0,C 180,E1 9223.481,E2 9223.481} C_VEL
LIN {X 0,Y 228.985,Z 936.993,A -85,B 0,C 180,E1 9221.32,E2 9221.32} C_VEL
LIN {X 0,Y 234.854,Z 920.64,A -85,B 0,C 180,E1 9219.594,E2 9219.594} C_VEL
LIN {X 0,Y 239.629,Z 904.324,A -85,B 0,C 180,E1 9218.332,E2 9218.332} C_VEL
LIN {X 0,Y 243.489,Z 886.602,A -85,B 0,C 180,E1 9217.348,E2 9217.348} C_VEL
LIN {X 0,Y 245.946,Z 868.472,A -85,B 0,C 180,E1 9216.672,E2 9216.672} C_VEL
LIN {X 0,Y 255.315,Z 746.486,A -85,B 0,C 180,E1 9213.516,E2 9213.516} C_VEL
LIN {X 0,Y 249.723,Z 736.148,A -85,B 0,C 180,E1 9210.696,E2 9210.696} C_VEL
LIN {X 0,Y 245.095,Z 728.447,A -85,B 0,C 180,E1 9208.044,E2 9208.044} C_VEL
LIN {X 0,Y 239.697,Z 720.249,A -85,B 0,C 180,E1 9204.456,E2 9204.456} C_VEL
LIN {X 0,Y 235.252,Z 714.032,A -85,B 0,C 180,E1 9200.786,E2 9200.786} C_VEL
LIN {X 0,Y 231.602,Z 709.459,A -85,B 0,C 180,E1 9196.942,E2 9196.942} C_VEL
LIN {X 0,Y 228.521,Z 705.668,A -85,B 0,C 180,E1 9192.123,E2 9192.123} C_VEL
LIN {X 0,Y 226.805,Z 704.387,A -85,B 0,C 180,E1 9186.327,E2 9186.327} C_VEL
LIN {X 0,Y 227.023,Z 705.012,A -85,B 0,C 180,E1 9181.766,E2 9181.766} C_VEL
LIN {X 0,Y 229.242,Z 708.755,A -85,B 0,C 180,E1 9175.873,E2 9175.873} C_VEL
LIN {X 0,Y 231.365,Z 712.366,A -85,B 0,C 180,E1 9172.675,E2 9172.675} C_VEL
LIN {X 0,Y 235.114,Z 718.207,A -85,B 0,C 180,E1 9168.656,E2 9168.656} C_VEL
LIN {X 0,Y 239.315,Z 725.461,A -85,B 0,C 180,E1 9165.11,E2 9165.11} C_VEL
LIN {X 0,Y 243,Z 732.194,A -85,B 0,C 180,E1 9162.52,E2 9162.52} C_VEL
LIN {X 0,Y 247.036,Z 740.132,A -85,B 0,C 180,E1 9160,E2 9160} C_VEL
LIN {X 0,Y 249.551,Z 745.855,A -85,B 0,C 180,E1 9158.539,E2 9158.539} C_VEL
LIN {X 0,Y 251.534,Z 770.703,A -85,B 0,C 180,E1 9156.273,E2 9156.273} C_VEL
LIN {X 0,Y 245.006,Z 849.356,A -85,B 0,C 180,E1 9154.076,E2 9154.076} C_VEL
LIN {X 0,Y 242.726,Z 865.758,A -85,B 0,C 180,E1 9153.25,E2 9153.25} C_VEL
LIN {X 0,Y 239.384,Z 881.651,A -85,B 0,C 180,E1 9152.08,E2 9152.08} C_VEL
LIN {X 0,Y 235.243,Z 896.271,A -85,B 0,C 180,E1 9150.611,E2 9150.611} C_VEL
LIN {X 0,Y 230.319,Z 910.032,A -85,B 0,C 180,E1 9148.783,E2 9148.783} C_VEL
LIN {X 0,Y 224.65,Z 923.212,A -85,B 0,C 180,E1 9146.502,E2 9146.502} C_VEL
LIN {X 0,Y 218.724,Z 934.841,A -85,B 0,C 180,E1 9143.863,E2 9143.863} C_VEL
LIN {X 0,Y 212.776,Z 945.049,A -85,B 0,C 180,E1 9140.837,E2 9140.837} C_VEL
LIN {X 0,Y 206.812,Z 954.083,A -85,B 0,C 180,E1 9137.295,E2 9137.295} C_VEL
LIN {X 0,Y 201.218,Z 961.489,A -85,B 0,C 180,E1 9133.292,E2 9133.292} C_VEL
LIN {X 0,Y 196.269,Z 967.324,A -85,B 0,C 180,E1 9128.79,E2 9128.79} C_VEL
LIN {X 0,Y 192.452,Z 971.103,A -85,B 0,C 180,E1 9124.132,E2 9124.132} C_VEL
LIN {X 0,Y 189.62,Z 973.223,A -85,B 0,C 180,E1 9119.019,E2 9119.019} C_VEL
LIN {X 0,Y 188.063,Z 973.44,A -85,B 0,C 180,E1 9114.165,E2 9114.165} C_VEL
LIN {X 0,Y 187.442,Z 971.911,A -85,B 0,C 180,E1 9108.989,E2 9108.989} C_VEL
LIN {X 0,Y 187.744,Z 968.844,A -85,B 0,C 180,E1 9104.18,E2 9104.18} C_VEL
LIN {X 0,Y 189.008,Z 963.646,A -85,B 0,C 180,E1 9099.131,E2 9099.131} C_VEL
LIN {X 0,Y 191.145,Z 956.897,A -85,B 0,C 180,E1 9094.5,E2 9094.5} C_VEL
LIN {X 0,Y 193.986,Z 948.58,A -85,B 0,C 180,E1 9090.295,E2 9090.295} C_VEL
LIN {X 0,Y 197.355,Z 938.885,A -85,B 0,C 180,E1 9086.514,E2 9086.514} C_VEL
LIN {X 0,Y 201.033,Z 927.685,A -85,B 0,C 180,E1 9083.144,E2 9083.144} C_VEL
LIN {X 0,Y 204.842,Z 915.011,A -85,B 0,C 180,E1 9080.163,E2 9080.163} C_VEL
LIN {X 0,Y 208.494,Z 901.256,A -85,B 0,C 180,E1 9077.677,E2 9077.677} C_VEL
LIN {X 0,Y 211.761,Z 886.59,A -85,B 0,C 180,E1 9075.647,E2 9075.647} C_VEL
LIN {X 0,Y 214.396,Z 871.63,A -85,B 0,C 180,E1 9074.098,E2 9074.098} C_VEL
LIN {X 0,Y 216.555,Z 854.2,A -85,B 0,C 180,E1 9072.838,E2 9072.838} C_VEL
LIN {X 0,Y 217.775,Z 836.757,A -85,B 0,C 180,E1 9072.071,E2 9072.071} C_VEL
LIN {X 0,Y 222.215,Z 760.46,A -85,B 0,C 180,E1 9069.699,E2 9069.699} C_VEL
LIN {X 0,Y 216.879,Z 713.198,A -85,B 0,C 180,E1 9066.472,E2 9066.472} C_VEL
LIN {X 0,Y 212.184,Z 703.328,A -85,B 0,C 180,E1 9064.791,E2 9064.791} C_VEL
LIN {X 0,Y 209.728,Z 691.767,A -85,B 0,C 180,E1 9060.19,E2 9060.19} C_VEL
LIN {X 0,Y 207.034,Z 681.303,A -85,B 0,C 180,E1 9055.426,E2 9055.426} C_VEL
LIN {X 0,Y 204.268,Z 672.323,A -85,B 0,C 180,E1 9050.66,E2 9050.66} C_VEL
LIN {X 0,Y 201.863,Z 665.231,A -85,B 0,C 180,E1 9046.317,E2 9046.317} C_VEL
LIN {X 0,Y 199.354,Z 658.567,A -85,B 0,C 180,E1 9041.457,E2 9041.457} C_VEL
LIN {X 0,Y 197.533,Z 654.385,A -85,B 0,C 180,E1 9037.769,E2 9037.769} C_VEL
LIN {X 0,Y 196.081,Z 650.782,A -85,B 0,C 180,E1 9034.12,E2 9034.12} C_VEL
LIN {X 0,Y 194.313,Z 646.753,A -85,B 0,C 180,E1 9028.927,E2 9028.927} C_VEL
LIN {X 0,Y 192.472,Z 642.665,A -85,B 0,C 180,E1 9020.369,E2 9020.369} C_VEL
LIN {X 0,Y 191.838,Z 641.857,A -85,B 0,C 180,E1 9014.18,E2 9014.18} C_VEL
LIN {X 0,Y 192.256,Z 642.339,A -85,B 0,C 180,E1 9007.772,E2 9007.772} C_VEL
LIN {X 0,Y 192.792,Z 643.49,A -85,B 0,C 180,E1 9004.164,E2 9004.164} C_VEL
LIN {X 0,Y 195.07,Z 647.864,A -85,B 0,C 180,E1 8996.18,E2 8996.18} C_VEL
LIN {X 0,Y 197.197,Z 652.42,A -85,B 0,C 180,E1 8990.957,E2 8990.957} C_VEL
LIN {X 0,Y 199.224,Z 656.897,A -85,B 0,C 180,E1 8986.948,E2 8986.948} C_VEL
LIN {X 0,Y 201.287,Z 661.86,A -85,B 0,C 180,E1 8983.256,E2 8983.256} C_VEL
LIN {X 0,Y 203.715,Z 667.403,A -85,B 0,C 180,E1 8979.606,E2 8979.606} C_VEL
LIN {X 0,Y 207.419,Z 677.157,A -85,B 0,C 180,E1 8974.348,E2 8974.348} C_VEL
LIN {X 0,Y 211.014,Z 687.77,A -85,B 0,C 180,E1 8969.586,E2 8969.586} C_VEL
LIN {X 0,Y 214.013,Z 697.634,A -85,B 0,C 180,E1 8965.787,E2 8965.787} C_VEL
LIN {X 0,Y 221.925,Z 712.577,A -85,B 0,C 180,E1 8963.146,E2 8963.146} C_VEL
LIN {X 0,Y 226.003,Z 720.864,A -85,B 0,C 180,E1 8961.912,E2 8961.912} C_VEL
LIN {X 0,Y 226.976,Z 724.785,A -85,B 0,C 180,E1 8961.548,E2 8961.548} C_VEL
LIN {X 0,Y 226.874,Z 730.176,A -85,B 0,C 180,E1 8961.348,E2 8961.348} C_VEL
LIN {X 0,Y 225.212,Z 737.837,A -85,B 0,C 180,E1 8961.377,E2 8961.377} C_VEL
LIN {X 0,Y 221.259,Z 751.619,A -85,B 0,C 180,E1 8961.636,E2 8961.636} C_VEL
LIN {X 0,Y 220.642,Z 756.32,A -85,B 0,C 180,E1 8961.571,E2 8961.571} C_VEL
LIN {X 0,Y 213.624,Z 875.18,A -85,B 0,C 180,E1 8958.078,E2 8958.078} C_VEL
LIN {X 0,Y 211.45,Z 893.38,A -85,B 0,C 180,E1 8957.12,E2 8957.12} C_VEL
LIN {X 0,Y 208.253,Z 910.776,A -85,B 0,C 180,E1 8955.782,E2 8955.782} C_VEL
LIN {X 0,Y 204.36,Z 927.357,A -85,B 0,C 180,E1 8954.009,E2 8954.009} C_VEL
LIN {X 0,Y 199.898,Z 943.387,A -85,B 0,C 180,E1 8951.702,E2 8951.702} C_VEL
LIN {X 0,Y 195.167,Z 958.477,A -85,B 0,C 180,E1 8948.858,E2 8948.858} C_VEL
LIN {X 0,Y 190.58,Z 972.009,A -85,B 0,C 180,E1 8945.592,E2 8945.592} C_VEL
LIN {X 0,Y 186.259,Z 984.549,A -85,B 0,C 180,E1 8941.742,E2 8941.742} C_VEL
LIN {X 0,Y 182.577,Z 995.713,A -85,B 0,C 180,E1 8937.389,E2 8937.389} C_VEL
LIN {X 0,Y 179.791,Z 1005.38,A -85,B 0,C 180,E1 8932.565,E2 8932.565} C_VEL
LIN {X 0,Y 178.122,Z 1013.548,A -85,B 0,C 180,E1 8927.309,E2 8927.309} C_VEL
LIN {X 0,Y 177.734,Z 1020.135,A -85,B 0,C 180,E1 8921.685,E2 8921.685} C_VEL
LIN {X 0,Y 178.401,Z 1024.506,A -85,B 0,C 180,E1 8916.437,E2 8916.437} C_VEL
LIN {X 0,Y 179.293,Z 1026.892,A -85,B 0,C 180,E1 8911.918,E2 8911.918} C_VEL
LIN {X 0,Y 179.335,Z 1027.65,A -85,B 0,C 180,E1 8909.042,E2 8909.042} C_VEL
LIN {X 0,Y 178.382,Z 1027.718,A -85,B 0,C 180,E1 8904.855,E2 8904.855} C_VEL
LIN {X 0,Y 177.373,Z 1026.215,A -85,B 0,C 180,E1 8899.28,E2 8899.28} C_VEL
LIN {X 0,Y 177.626,Z 1022.852,A -85,B 0,C 180,E1 8893.317,E2 8893.317} C_VEL
LIN {X 0,Y 179.58,Z 1017.666,A -85,B 0,C 180,E1 8887.408,E2 8887.408} C_VEL
LIN {X 0,Y 183.386,Z 1010.567,A -85,B 0,C 180,E1 8881.684,E2 8881.684} C_VEL
LIN {X 0,Y 188.64,Z 1001.916,A -85,B 0,C 180,E1 8876.549,E2 8876.549} C_VEL
LIN {X 0,Y 194.979,Z 991.685,A -85,B 0,C 180,E1 8872.022,E2 8872.022} C_VEL
LIN {X 0,Y 201.587,Z 980.774,A -85,B 0,C 180,E1 8868.346,E2 8868.346} C_VEL
LIN {X 0,Y 209.079,Z 967.544,A -85,B 0,C 180,E1 8864.947,E2 8864.947} C_VEL
LIN {X 0,Y 216.133,Z 953.782,A -85,B 0,C 180,E1 8862.254,E2 8862.254} C_VEL
LIN {X 0,Y 222.774,Z 939.171,A -85,B 0,C 180,E1 8860.072,E2 8860.072} C_VEL
LIN {X 0,Y 228.793,Z 923.635,A -85,B 0,C 180,E1 8858.332,E2 8858.332} C_VEL
LIN {X 0,Y 234.04,Z 907.143,A -85,B 0,C 180,E1 8856.975,E2 8856.975} C_VEL
LIN {X 0,Y 238.38,Z 889.104,A -85,B 0,C 180,E1 8855.913,E2 8855.913} C_VEL
LIN {X 0,Y 241.228,Z 871.103,A -85,B 0,C 180,E1 8855.186,E2 8855.186} C_VEL
LIN {X 0,Y 250.904,Z 750.384,A -85,B 0,C 180,E1 8852.039,E2 8852.039} C_VEL
LIN {X 0,Y 245.511,Z 740.198,A -85,B 0,C 180,E1 8849.055,E2 8849.055} C_VEL
LIN {X 0,Y 240.511,Z 731.984,A -85,B 0,C 180,E1 8845.881,E2 8845.881} C_VEL
LIN {X 0,Y 236.816,Z 726.225,A -85,B 0,C 180,E1 8843.119,E2 8843.119} C_VEL
LIN {X 0,Y 233.483,Z 721.458,A -85,B 0,C 180,E1 8840.165,E2 8840.165} C_VEL
LIN {X 0,Y 230.123,Z 717.047,A -85,B 0,C 180,E1 8836.404,E2 8836.404} C_VEL
LIN {X 0,Y 227.392,Z 713.552,A -85,B 0,C 180,E1 8831.926,E2 8831.926} C_VEL
LIN {X 0,Y 225.764,Z 712.316,A -85,B 0,C 180,E1 8826.101,E2 8826.101} C_VEL
LIN {X 0,Y 225.955,Z 712.874,A -85,B 0,C 180,E1 8822.028,E2 8822.028} C_VEL
LIN {X 0,Y 228.058,Z 716.648,A -85,B 0,C 180,E1 8816.103,E2 8816.103} C_VEL
LIN {X 0,Y 229.94,Z 720.043,A -85,B 0,C 180,E1 8813.132,E2 8813.132} C_VEL
LIN {X 0,Y 233.35,Z 725.651,A -85,B 0,C 180,E1 8809.257,E2 8809.257} C_VEL
LIN {X 0,Y 237.24,Z 732.684,A -85,B 0,C 180,E1 8805.788,E2 8805.788} C_VEL
LIN {X 0,Y 240.612,Z 739.167,A -85,B 0,C 180,E1 8803.275,E2 8803.275} C_VEL
LIN {X 0,Y 244.723,Z 747.587,A -85,B 0,C 180,E1 8800.581,E2 8800.581} C_VEL
LIN {X 0,Y 245.904,Z 750.831,A -85,B 0,C 180,E1 8799.811,E2 8799.811} C_VEL
LIN {X 0,Y 247.34,Z 772.437,A -85,B 0,C 180,E1 8797.815,E2 8797.815} C_VEL
LIN {X 0,Y 240.656,Z 850.016,A -85,B 0,C 180,E1 8795.653,E2 8795.653} C_VEL
LIN {X 0,Y 238.263,Z 866.543,A -85,B 0,C 180,E1 8794.821,E2 8794.821} C_VEL
LIN {X 0,Y 234.686,Z 882.838,A -85,B 0,C 180,E1 8793.618,E2 8793.618} C_VEL
LIN {X 0,Y 230.179,Z 897.919,A -85,B 0,C 180,E1 8792.085,E2 8792.085} C_VEL
LIN {X 0,Y 224.652,Z 912.531,A -85,B 0,C 180,E1 8790.1,E2 8790.1} C_VEL
LIN {X 0,Y 218.974,Z 924.968,A -85,B 0,C 180,E1 8787.888,E2 8787.888} C_VEL
LIN {X 0,Y 212.516,Z 936.892,A -85,B 0,C 180,E1 8785.1,E2 8785.1} C_VEL
LIN {X 0,Y 205.983,Z 947.417,A -85,B 0,C 180,E1 8781.846,E2 8781.846} C_VEL
LIN {X 0,Y 199.764,Z 956.101,A -85,B 0,C 180,E1 8778.225,E2 8778.225} C_VEL
LIN {X 0,Y 193.933,Z 963.316,A -85,B 0,C 180,E1 8774.108,E2 8774.108} C_VEL
LIN {X 0,Y 189.072,Z 968.627,A -85,B 0,C 180,E1 8769.782,E2 8769.782} C_VEL
LIN {X 0,Y 184.984,Z 972.372,A -85,B 0,C 180,E1 8764.955,E2 8764.955} C_VEL
LIN {X 0,Y 181.931,Z 974.462,A -85,B 0,C 180,E1 8759.644,E2 8759.644} C_VEL
LIN {X 0,Y 180.149,Z 974.6,A -85,B 0,C 180,E1 8754.249,E2 8754.249} C_VEL
LIN {X 0,Y 179.515,Z 972.922,A -85,B 0,C 180,E1 8748.76,E2 8748.76} C_VEL
LIN {X 0,Y 179.917,Z 969.421,A -85,B 0,C 180,E1 8743.456,E2 8743.456} C_VEL
LIN {X 0,Y 181.36,Z 964.054,A -85,B 0,C 180,E1 8738.241,E2 8738.241} C_VEL
LIN {X 0,Y 183.528,Z 957.536,A -85,B 0,C 180,E1 8733.748,E2 8733.748} C_VEL
LIN {X 0,Y 186.563,Z 949.115,A -85,B 0,C 180,E1 8729.385,E2 8729.385} C_VEL
LIN {X 0,Y 190.138,Z 939.281,A -85,B 0,C 180,E1 8725.475,E2 8725.475} C_VEL
LIN {X 0,Y 194.2,Z 927.406,A -85,B 0,C 180,E1 8721.86,E2 8721.86} C_VEL
LIN {X 0,Y 198.048,Z 915.1,A -85,B 0,C 180,E1 8718.939,E2 8718.939} C_VEL
LIN {X 0,Y 201.881,Z 901.101,A -85,B 0,C 180,E1 8716.393,E2 8716.393} C_VEL
LIN {X 0,Y 205.309,Z 886.199,A -85,B 0,C 180,E1 8714.318,E2 8714.318} C_VEL
LIN {X 0,Y 208.058,Z 870.734,A -85,B 0,C 180,E1 8712.737,E2 8712.737} C_VEL
LIN {X 0,Y 210.195,Z 853.807,A -85,B 0,C 180,E1 8711.522,E2 8711.522} C_VEL
LIN {X 0,Y 211.506,Z 834.704,A -85,B 0,C 180,E1 8710.711,E2 8710.711} C_VEL
LIN {X 0,Y 215.965,Z 761.5,A -85,B 0,C 180,E1 8708.403,E2 8708.403} C_VEL
LIN {X 0,Y 211.236,Z 716.971,A -85,B 0,C 180,E1 8705.262,E2 8705.262} C_VEL
LIN {X 0,Y 204.645,Z 703.254,A -85,B 0,C 180,E1 8702.777,E2 8702.777} C_VEL
LIN {X 0,Y 202.407,Z 693.02,A -85,B 0,C 180,E1 8698.423,E2 8698.423} C_VEL
LIN {X 0,Y 200.028,Z 683.644,A -85,B 0,C 180,E1 8693.854,E2 8693.854} C_VEL
LIN {X 0,Y 197.402,Z 675.109,A -85,B 0,C 180,E1 8689,E2 8689} C_VEL
LIN {X 0,Y 194.92,Z 667.583,A -85,B 0,C 180,E1 8683.977,E2 8683.977} C_VEL
LIN {X 0,Y 192.792,Z 662.29,A -85,B 0,C 180,E1 8679.637,E2 8679.637} C_VEL
LIN {X 0,Y 191.74,Z 659.725,A -85,B 0,C 180,E1 8677.223,E2 8677.223} C_VEL
LIN {X 0,Y 190.504,Z 656.458,A -85,B 0,C 180,E1 8673.804,E2 8673.804} C_VEL
LIN {X 0,Y 188.934,Z 652.658,A -85,B 0,C 180,E1 8668.79,E2 8668.79} C_VEL
LIN {X 0,Y 187.261,Z 648.735,A -85,B 0,C 180,E1 8660.308,E2 8660.308} C_VEL
LIN {X 0,Y 186.672,Z 647.979,A -85,B 0,C 180,E1 8653.948,E2 8653.948} C_VEL
LIN {X 0,Y 187.18,Z 648.554,A -85,B 0,C 180,E1 8647.366,E2 8647.366} C_VEL
LIN {X 0,Y 187.683,Z 649.876,A -85,B 0,C 180,E1 8643.666,E2 8643.666} C_VEL
LIN {X 0,Y 189.759,Z 653.844,A -85,B 0,C 180,E1 8636.375,E2 8636.375} C_VEL
LIN {X 0,Y 191.735,Z 658.157,A -85,B 0,C 180,E1 8631.302,E2 8631.302} C_VEL
LIN {X 0,Y 193.687,Z 662.674,A -85,B 0,C 180,E1 8627.175,E2 8627.175} C_VEL
LIN {X 0,Y 195.726,Z 667.662,A -85,B 0,C 180,E1 8623.378,E2 8623.378} C_VEL
LIN {X 0,Y 197.907,Z 672.858,A -85,B 0,C 180,E1 8619.907,E2 8619.907} C_VEL
LIN {X 0,Y 201.353,Z 682.22,A -85,B 0,C 180,E1 8614.72,E2 8614.72} C_VEL
LIN {X 0,Y 204.617,Z 692.204,A -85,B 0,C 180,E1 8610.105,E2 8610.105} C_VEL
LIN {X 0,Y 206.599,Z 698.557,A -85,B 0,C 180,E1 8607.631,E2 8607.631} C_VEL
LIN {X 0,Y 214.994,Z 713.98,A -85,B 0,C 180,E1 8604.702,E2 8604.702} C_VEL
LIN {X 0,Y 220.914,Z 726.42,A -85,B 0,C 180,E1 8602.777,E2 8602.777} C_VEL
LIN {X 0,Y 221.474,Z 742.942,A -85,B 0,C 180,E1 8601.953,E2 8601.953} C_VEL
LIN {X 0,Y 220.642,Z 756.32,A -85,B 0,C 180,E1 8601.571,E2 8601.571} C_VEL
LIN {X 0,Y 219.418,Z 763.985,A -85,B 0,C 180,E1 8601.511,E2 8601.511} C_VEL
LIN {X 0,Y 213.297,Z 784.265,A -85,B 0,C 180,E1 8601.984,E2 8601.984} C_VEL
LIN {X 0,Y 212.329,Z 790.849,A -85,B 0,C 180,E1 8601.917,E2 8601.917} C_VEL
LIN {X 0,Y 207.207,Z 874.639,A -85,B 0,C 180,E1 8599.384,E2 8599.384} C_VEL
LIN {X 0,Y 204.953,Z 892.821,A -85,B 0,C 180,E1 8598.407,E2 8598.407} C_VEL
LIN {X 0,Y 201.591,Z 910.445,A -85,B 0,C 180,E1 8597.02,E2 8597.02} C_VEL
LIN {X 0,Y 197.439,Z 927.394,A -85,B 0,C 180,E1 8595.153,E2 8595.153} C_VEL
LIN {X 0,Y 192.82,Z 943.232,A -85,B 0,C 180,E1 8592.79,E2 8592.79} C_VEL
LIN {X 0,Y 187.902,Z 958.243,A -85,B 0,C 180,E1 8589.859,E2 8589.859} C_VEL
LIN {X 0,Y 182.976,Z 972.117,A -85,B 0,C 180,E1 8586.363,E2 8586.363} C_VEL
LIN {X 0,Y 178.331,Z 984.972,A -85,B 0,C 180,E1 8582.185,E2 8582.185} C_VEL
LIN {X 0,Y 174.569,Z 995.811,A -85,B 0,C 180,E1 8577.642,E2 8577.642} C_VEL
LIN {X 0,Y 171.747,Z 1005.245,A -85,B 0,C 180,E1 8572.597,E2 8572.597} C_VEL
LIN {X 0,Y 170.107,Z 1013.205,A -85,B 0,C 180,E1 8567.092,E2 8567.092} C_VEL
LIN {X 0,Y 169.793,Z 1019.258,A -85,B 0,C 180,E1 8561.55,E2 8561.55} C_VEL
LIN {X 0,Y 170.533,Z 1023.533,A -85,B 0,C 180,E1 8556.059,E2 8556.059} C_VEL
LIN {X 0,Y 171.413,Z 1025.696,A -85,B 0,C 180,E1 8551.672,E2 8551.672} C_VEL
LIN {X 0,Y 171.367,Z 1026.429,A -85,B 0,C 180,E1 8548.663,E2 8548.663} C_VEL
LIN {X 0,Y 170.223,Z 1026.394,A -85,B 0,C 180,E1 8543.931,E2 8543.931} C_VEL
LIN {X 0,Y 169.34,Z 1024.605,A -85,B 0,C 180,E1 8537.728,E2 8537.728} C_VEL
LIN {X 0,Y 170.116,Z 1020.772,A -85,B 0,C 180,E1 8531.133,E2 8531.133} C_VEL
LIN {X 0,Y 172.777,Z 1015.299,A -85,B 0,C 180,E1 8525.011,E2 8525.011} C_VEL
LIN {X 0,Y 177.063,Z 1008.325,A -85,B 0,C 180,E1 8519.455,E2 8519.455} C_VEL
LIN {X 0,Y 183.007,Z 999.336,A -85,B 0,C 180,E1 8514.226,E2 8514.226} C_VEL
LIN {X 0,Y 190.003,Z 988.779,A -85,B 0,C 180,E1 8509.665,E2 8509.665} C_VEL
LIN {X 0,Y 197.733,Z 976.661,A -85,B 0,C 180,E1 8505.749,E2 8505.749} C_VEL
LIN {X 0,Y 205.48,Z 963.426,A -85,B 0,C 180,E1 8502.528,E2 8502.528} C_VEL
LIN {X 0,Y 213.031,Z 948.901,A -85,B 0,C 180,E1 8499.881,E2 8499.881} C_VEL
LIN {X 0,Y 220.064,Z 933.343,A -85,B 0,C 180,E1 8497.762,E2 8497.762} C_VEL
LIN {X 0,Y 226.055,Z 917.618,A -85,B 0,C 180,E1 8496.176,E2 8496.176} C_VEL
LIN {X 0,Y 231.155,Z 900.934,A -85,B 0,C 180,E1 8494.947,E2 8494.947} C_VEL
LIN {X 0,Y 235.067,Z 883.242,A -85,B 0,C 180,E1 8494.028,E2 8494.028} C_VEL
LIN {X 0,Y 237.592,Z 864.638,A -85,B 0,C 180,E1 8493.376,E2 8493.376} C_VEL
LIN {X 0,Y 246.714,Z 754.316,A -85,B 0,C 180,E1 8490.532,E2 8490.532} C_VEL
LIN {X 0,Y 241.761,Z 744.924,A -85,B 0,C 180,E1 8487.527,E2 8487.527} C_VEL
LIN {X 0,Y 237.939,Z 738.525,A -85,B 0,C 180,E1 8484.914,E2 8484.914} C_VEL
LIN {X 0,Y 234.81,Z 733.417,A -85,B 0,C 180,E1 8482.402,E2 8482.402} C_VEL
LIN {X 0,Y 231.742,Z 728.882,A -85,B 0,C 180,E1 8479.534,E2 8479.534} C_VEL
LIN {X 0,Y 228.753,Z 724.749,A -85,B 0,C 180,E1 8475.983,E2 8475.983} C_VEL
LIN {X 0,Y 226.152,Z 721.346,A -85,B 0,C 180,E1 8471.475,E2 8471.475} C_VEL
LIN {X 0,Y 224.726,Z 720.248,A -85,B 0,C 180,E1 8465.873,E2 8465.873} C_VEL
LIN {X 0,Y 224.924,Z 720.886,A -85,B 0,C 180,E1 8462.038,E2 8462.038} C_VEL
LIN {X 0,Y 226.811,Z 724.424,A -85,B 0,C 180,E1 8456.461,E2 8456.461} C_VEL
LIN {X 0,Y 228.531,Z 727.717,A -85,B 0,C 180,E1 8453.594,E2 8453.594} C_VEL
LIN {X 0,Y 231.613,Z 733.091,A -85,B 0,C 180,E1 8449.868,E2 8449.868} C_VEL
LIN {X 0,Y 235.213,Z 739.906,A -85,B 0,C 180,E1 8446.479,E2 8446.479} C_VEL
LIN {X 0,Y 238.265,Z 746.134,A -85,B 0,C 180,E1 8444.045,E2 8444.045} C_VEL
LIN {X 0,Y 241.982,Z 754.217,A -85,B 0,C 180,E1 8441.448,E2 8441.448} C_VEL
LIN {X 0,Y 242.403,Z 755.858,A -85,B 0,C 180,E1 8441.122,E2 8441.122} C_VEL
LIN {X 0,Y 243.364,Z 774.133,A -85,B 0,C 180,E1 8439.415,E2 8439.415} C_VEL
LIN {X 0,Y 236.497,Z 850.694,A -85,B 0,C 180,E1 8437.286,E2 8437.286} C_VEL
LIN {X 0,Y 234.008,Z 867.218,A -85,B 0,C 180,E1 8436.458,E2 8436.458} C_VEL
LIN {X 0,Y 230.352,Z 883.292,A -85,B 0,C 180,E1 8435.281,E2 8435.281} C_VEL
LIN {X 0,Y 225.721,Z 898.337,A -85,B 0,C 180,E1 8433.77,E2 8433.77} C_VEL
LIN {X 0,Y 219.934,Z 913.09,A -85,B 0,C 180,E1 8431.783,E2 8431.783} C_VEL
LIN {X 0,Y 213.657,Z 926.261,A -85,B 0,C 180,E1 8429.437,E2 8429.437} C_VEL
LIN {X 0,Y 207.012,Z 937.965,A -85,B 0,C 180,E1 8426.676,E2 8426.676} C_VEL
LIN {X 0,Y 200.311,Z 948.234,A -85,B 0,C 180,E1 8423.478,E2 8423.478} C_VEL
LIN {X 0,Y 193.725,Z 956.999,A -85,B 0,C 180,E1 8419.805,E2 8419.805} C_VEL
LIN {X 0,Y 187.5,Z 964.258,A -85,B 0,C 180,E1 8415.607,E2 8415.607} C_VEL
LIN {X 0,Y 182.264,Z 969.632,A -85,B 0,C 180,E1 8411.169,E2 8411.169} C_VEL
LIN {X 0,Y 177.81,Z 973.452,A -85,B 0,C 180,E1 8406.187,E2 8406.187} C_VEL
LIN {X 0,Y 174.424,Z 975.613,A -85,B 0,C 180,E1 8400.675,E2 8400.675} C_VEL
LIN {X 0,Y 172.448,Z 975.89,A -85,B 0,C 180,E1 8395.243,E2 8395.243} C_VEL
LIN {X 0,Y 171.607,Z 974.294,A -85,B 0,C 180,E1 8389.396,E2 8389.396} C_VEL
LIN {X 0,Y 171.875,Z 971.2,A -85,B 0,C 180,E1 8384.142,E2 8384.142} C_VEL
LIN {X 0,Y 173.228,Z 965.993,A -85,B 0,C 180,E1 8378.63,E2 8378.63} C_VEL
LIN {X 0,Y 175.56,Z 959.26,A -85,B 0,C 180,E1 8373.591,E2 8373.591} C_VEL
LIN {X 0,Y 178.67,Z 950.978,A -85,B 0,C 180,E1 8369.037,E2 8369.037} C_VEL
LIN {X 0,Y 182.355,Z 941.331,A -85,B 0,C 180,E1 8364.966,E2 8364.966} C_VEL
LIN {X 0,Y 186.38,Z 930.253,A -85,B 0,C 180,E1 8361.36,E2 8361.36} C_VEL
LIN {X 0,Y 190.734,Z 917.074,A -85,B 0,C 180,E1 8358.049,E2 8358.049} C_VEL
LIN {X 0,Y 194.72,Z 903.403,A -85,B 0,C 180,E1 8355.427,E2 8355.427} C_VEL
LIN {X 0,Y 198.442,Z 888.126,A -85,B 0,C 180,E1 8353.204,E2 8353.204} C_VEL
LIN {X 0,Y 201.354,Z 872.934,A -85,B 0,C 180,E1 8351.566,E2 8351.566} C_VEL
LIN {X 0,Y 203.715,Z 855.413,A -85,B 0,C 180,E1 8350.251,E2 8350.251} C_VEL
LIN {X 0,Y 205.065,Z 837.776,A -85,B 0,C 180,E1 8349.447,E2 8349.447} C_VEL
LIN {X 0,Y 209.827,Z 762.48,A -85,B 0,C 180,E1 8347.026,E2 8347.026} C_VEL
LIN {X 0,Y 205.611,Z 720.509,A -85,B 0,C 180,E1 8343.952,E2 8343.952} C_VEL
LIN {X 0,Y 199.293,Z 707.46,A -85,B 0,C 180,E1 8341.477,E2 8341.477} C_VEL
LIN {X 0,Y 197.055,Z 702.715,A -85,B 0,C 180,E1 8340.39,E2 8340.39} C_VEL
LIN {X 0,Y 194.623,Z 691.867,A -85,B 0,C 180,E1 8335.285,E2 8335.285} C_VEL
LIN {X 0,Y 192.305,Z 683.397,A -85,B 0,C 180,E1 8330.629,E2 8330.629} C_VEL
LIN {X 0,Y 189.876,Z 675.517,A -85,B 0,C 180,E1 8325.543,E2 8325.543} C_VEL
LIN {X 0,Y 187.624,Z 669.129,A -85,B 0,C 180,E1 8320.554,E2 8320.554} C_VEL
LIN {X 0,Y 186.136,Z 665.38,A -85,B 0,C 180,E1 8316.987,E2 8316.987} C_VEL
LIN {X 0,Y 184.946,Z 662.14,A -85,B 0,C 180,E1 8313.466,E2 8313.466} C_VEL
LIN {X 0,Y 183.453,Z 658.416,A -85,B 0,C 180,E1 8308.306,E2 8308.306} C_VEL
LIN {X 0,Y 182.002,Z 654.727,A -85,B 0,C 180,E1 8299.915,E2 8299.915} C_VEL
LIN {X 0,Y 181.513,Z 654.105,A -85,B 0,C 180,E1 8293.702,E2 8293.702} C_VEL
LIN {X 0,Y 182.052,Z 654.702,A -85,B 0,C 180,E1 8287.258,E2 8287.258} C_VEL
LIN {X 0,Y 182.585,Z 656.273,A -85,B 0,C 180,E1 8283.14,E2 8283.14} C_VEL
LIN {X 0,Y 184.443,Z 659.817,A -85,B 0,C 180,E1 8276.582,E2 8276.582} C_VEL
LIN {X 0,Y 186.359,Z 664.236,A -85,B 0,C 180,E1 8271.361,E2 8271.361} C_VEL
LIN {X 0,Y 188.148,Z 668.437,A -85,B 0,C 180,E1 8267.416,E2 8267.416} C_VEL
LIN {X 0,Y 190.803,Z 674.785,A -85,B 0,C 180,E1 8262.506,E2 8262.506} C_VEL
LIN {X 0,Y 194.113,Z 683.833,A -85,B 0,C 180,E1 8256.955,E2 8256.955} C_VEL
LIN {X 0,Y 197.209,Z 693.239,A -85,B 0,C 180,E1 8252.197,E2 8252.197} C_VEL
LIN {X 0,Y 199.013,Z 698.806,A -85,B 0,C 180,E1 8249.841,E2 8249.841} C_VEL
LIN {X 0,Y 207.534,Z 714.13,A -85,B 0,C 180,E1 8246.604,E2 8246.604} C_VEL
LIN {X 0,Y 214.92,Z 729.212,A -85,B 0,C 180,E1 8244.032,E2 8244.032} C_VEL
LIN {X 0,Y 215.326,Z 743.756,A -85,B 0,C 180,E1 8243.289,E2 8243.289} C_VEL
LIN {X 0,Y 212.329,Z 790.849,A -85,B 0,C 180,E1 8241.917,E2 8241.917} C_VEL
LIN {X 0,Y 211.113,Z 798.514,A -85,B 0,C 180,E1 8241.859,E2 8241.859} C_VEL
LIN {X 0,Y 205.024,Z 818.799,A -85,B 0,C 180,E1 8242.362,E2 8242.362} C_VEL
LIN {X 0,Y 204.046,Z 825.384,A -85,B 0,C 180,E1 8242.3,E2 8242.3} C_VEL
LIN {X 0,Y 200.866,Z 874.467,A -85,B 0,C 180,E1 8240.757,E2 8240.757} C_VEL
LIN {X 0,Y 198.465,Z 892.864,A -85,B 0,C 180,E1 8239.737,E2 8239.737} C_VEL
LIN {X 0,Y 195.043,Z 910.056,A -85,B 0,C 180,E1 8238.347,E2 8238.347} C_VEL
LIN {X 0,Y 190.879,Z 926.401,A -85,B 0,C 180,E1 8236.511,E2 8236.511} C_VEL
LIN {X 0,Y 186.071,Z 942.264,A -85,B 0,C 180,E1 8234.098,E2 8234.098} C_VEL
LIN {X 0,Y 180.965,Z 957.203,A -85,B 0,C 180,E1 8231.11,E2 8231.11} C_VEL
LIN {X 0,Y 175.783,Z 971.153,A -85,B 0,C 180,E1 8227.491,E2 8227.491} C_VEL
LIN {X 0,Y 170.987,Z 983.761,A -85,B 0,C 180,E1 8223.26,E2 8223.26} C_VEL
LIN {X 0,Y 166.803,Z 995.183,A -85,B 0,C 180,E1 8218.266,E2 8218.266} C_VEL
LIN {X 0,Y 163.704,Z 1005.1,A -85,B 0,C 180,E1 8212.631,E2 8212.631} C_VEL
LIN {X 0,Y 162.093,Z 1012.86,A -85,B 0,C 180,E1 8206.854,E2 8206.854} C_VEL
LIN {X 0,Y 161.885,Z 1018.844,A -85,B 0,C 180,E1 8200.877,E2 8200.877} C_VEL
LIN {X 0,Y 162.745,Z 1022.772,A -85,B 0,C 180,E1 8195.288,E2 8195.288} C_VEL
LIN {X 0,Y 163.578,Z 1024.612,A -85,B 0,C 180,E1 8191.051,E2 8191.051} C_VEL
LIN {X 0,Y 163.294,Z 1025.238,A -85,B 0,C 180,E1 8187.895,E2 8187.895} C_VEL
LIN {X 0,Y 161.976,Z 1024.993,A -85,B 0,C 180,E1 8182.552,E2 8182.552} C_VEL
LIN {X 0,Y 161.401,Z 1022.99,A -85,B 0,C 180,E1 8176.02,E2 8176.02} C_VEL
LIN {X 0,Y 162.595,Z 1019.215,A -85,B 0,C 180,E1 8169.482,E2 8169.482} C_VEL
LIN {X 0,Y 165.814,Z 1013.622,A -85,B 0,C 180,E1 8163.112,E2 8163.112} C_VEL
LIN {X 0,Y 170.693,Z 1006.48,A -85,B 0,C 180,E1 8157.391,E2 8157.391} C_VEL
LIN {X 0,Y 176.938,Z 997.786,A -85,B 0,C 180,E1 8152.29,E2 8152.29} C_VEL
LIN {X 0,Y 184.356,Z 987.366,A -85,B 0,C 180,E1 8147.739,E2 8147.739} C_VEL
LIN {X 0,Y 191.985,Z 976.098,A -85,B 0,C 180,E1 8144.053,E2 8144.053} C_VEL
LIN {X 0,Y 200.121,Z 962.947,A -85,B 0,C 180,E1 8140.806,E2 8140.806} C_VEL
LIN {X 0,Y 207.948,Z 948.609,A -85,B 0,C 180,E1 8138.174,E2 8138.174} C_VEL
LIN {X 0,Y 215.235,Z 933.191,A -85,B 0,C 180,E1 8136.07,E2 8136.07} C_VEL
LIN {X 0,Y 221.419,Z 917.643,A -85,B 0,C 180,E1 8134.502,E2 8134.502} C_VEL
LIN {X 0,Y 226.861,Z 900.601,A -85,B 0,C 180,E1 8133.249,E2 8133.249} C_VEL
LIN {X 0,Y 230.911,Z 883.01,A -85,B 0,C 180,E1 8132.34,E2 8132.34} C_VEL
LIN {X 0,Y 233.548,Z 864.515,A -85,B 0,C 180,E1 8131.693,E2 8131.693} C_VEL
LIN {X 0,Y 242.72,Z 758.52,A -85,B 0,C 180,E1 8128.962,E2 8128.962} C_VEL
LIN {X 0,Y 238.66,Z 750.64,A -85,B 0,C 180,E1 8126.293,E2 8126.293} C_VEL
LIN {X 0,Y 235.394,Z 744.927,A -85,B 0,C 180,E1 8123.865,E2 8123.865} C_VEL
LIN {X 0,Y 232.708,Z 740.429,A -85,B 0,C 180,E1 8121.553,E2 8121.553} C_VEL
LIN {X 0,Y 230.03,Z 736.303,A -85,B 0,C 180,E1 8118.894,E2 8118.894} C_VEL
LIN {X 0,Y 227.31,Z 732.338,A -85,B 0,C 180,E1 8115.433,E2 8115.433} C_VEL
LIN {X 0,Y 225.041,Z 729.232,A -85,B 0,C 180,E1 8111.273,E2 8111.273} C_VEL
LIN {X 0,Y 223.712,Z 728.183,A -85,B 0,C 180,E1 8105.9,E2 8105.9} C_VEL
LIN {X 0,Y 223.861,Z 728.747,A -85,B 0,C 180,E1 8102.303,E2 8102.303} C_VEL
LIN {X 0,Y 225.573,Z 732.2,A -85,B 0,C 180,E1 8096.823,E2 8096.823} C_VEL
LIN {X 0,Y 227.137,Z 735.388,A -85,B 0,C 180,E1 8094.062,E2 8094.062} C_VEL
LIN {X 0,Y 229.851,Z 740.408,A -85,B 0,C 180,E1 8090.548,E2 8090.548} C_VEL
LIN {X 0,Y 233.219,Z 747.125,A -85,B 0,C 180,E1 8087.181,E2 8087.181} C_VEL
LIN {X 0,Y 236.247,Z 753.73,A -85,B 0,C 180,E1 8084.598,E2 8084.598} C_VEL
LIN {X 0,Y 239.005,Z 760.366,A -85,B 0,C 180,E1 8082.526,E2 8082.526} C_VEL
LIN {X 0,Y 239.614,Z 775.937,A -85,B 0,C 180,E1 8081.069,E2 8081.069} C_VEL
LIN {X 0,Y 232.599,Z 851.425,A -85,B 0,C 180,E1 8078.983,E2 8078.983} C_VEL
LIN {X 0,Y 230.008,Z 867.927,A -85,B 0,C 180,E1 8078.161,E2 8078.161} C_VEL
LIN {X 0,Y 226.21,Z 883.963,A -85,B 0,C 180,E1 8076.995,E2 8076.995} C_VEL
LIN {X 0,Y 221.473,Z 898.823,A -85,B 0,C 180,E1 8075.52,E2 8075.52} C_VEL
LIN {X 0,Y 215.503,Z 913.479,A -85,B 0,C 180,E1 8073.566,E2 8073.566} C_VEL
LIN {X 0,Y 209.156,Z 926.361,A -85,B 0,C 180,E1 8071.307,E2 8071.307} C_VEL
LIN {X 0,Y 202.486,Z 937.778,A -85,B 0,C 180,E1 8068.678,E2 8068.678} C_VEL
LIN {X 0,Y 195.043,Z 948.729,A -85,B 0,C 180,E1 8065.317,E2 8065.317} C_VEL
LIN {X 0,Y 188.359,Z 957.307,A -85,B 0,C 180,E1 8061.778,E2 8061.778} C_VEL
LIN {X 0,Y 181.652,Z 964.754,A -85,B 0,C 180,E1 8057.524,E2 8057.524} C_VEL
LIN {X 0,Y 175.574,Z 970.641,A -85,B 0,C 180,E1 8052.662,E2 8052.662} C_VEL
LIN {X 0,Y 170.73,Z 974.551,A -85,B 0,C 180,E1 8047.521,E2 8047.521} C_VEL
LIN {X 0,Y 166.954,Z 976.784,A -85,B 0,C 180,E1 8041.742,E2 8041.742} C_VEL
LIN {X 0,Y 164.684,Z 977.122,A -85,B 0,C 180,E1 8035.921,E2 8035.921} C_VEL
LIN {X 0,Y 163.702,Z 975.569,A -85,B 0,C 180,E1 8029.845,E2 8029.845} C_VEL
LIN {X 0,Y 163.94,Z 972.378,A -85,B 0,C 180,E1 8024.12,E2 8024.12} C_VEL
LIN {X 0,Y 165.344,Z 967.165,A -85,B 0,C 180,E1 8018.344,E2 8018.344} C_VEL
LIN {X 0,Y 167.787,Z 960.438,A -85,B 0,C 180,E1 8013.074,E2 8013.074} C_VEL
